// TIA Portal project "Divider LIE-09" (V14)

(* hardware
DEVICE "S7-1200 station"  S7-1200 Station
   slot 0: "Rack_0"  Rack  V1.0
   slot 1: "CLP_Divider"  CPU 1214C DC/DC/DC  6ES7 214-1AG40-0XB0  V4.1
   slot 2: "Analog_Output"  6ES7 232-4HD32-0XB0  V2.0
DEVICE "IHM_Divider"  KTP600 Basic mono PN
   slot 0: "HMI"  HMI  6AV6 647-0AB11-3AX0  12.0.0.0
   slot 1: "HMI_RT_2"  KTP600 Basic mono PN  6AV6 647-0AB11-3AX0  12.0.0.0
   slot 5: "IHM_Divider.IE_CP_1"  PROFINET Interface
      slot 1: "PROFINET Interface_1"  PROFINET Interface
         slot 1: "Port_1"  Port
*)

// ===== PLC "CLP_Divider"  CPU 1214C DC/DC/DC =====

VAR_GLOBAL   // PLC tag table "General"
   "Aux_Byte_0" AT %MB10 : Byte;
   "Aux_Byte_1" AT %MB11 : Byte;
   "Aux_Int" AT %MW10 : Int;
   "Aux_Real" AT %MD12 : Real;
   "Status Byte" AT %QB50 : Byte;   // Palavra de status enviada para a SteelBelt
END_VAR

VAR_GLOBAL   // PLC tag table "Digital Output"
   "DO - Ligar Inv 01" AT %Q0.0 : Bool;
   "DO - Ligar Inv 02" AT %Q0.1 : Bool;
   "DO - Reset Inv 01" AT %Q0.2 : Bool;
   "DO - Reset Inv 02" AT %Q0.3 : Bool;
   "DO - Ligar Inv Divider" AT %Q0.4 : Bool;
   "DO - Reserva 02" AT %Q0.5 : Bool;
   "DO - Reserva 03" AT %Q0.6 : Bool;
END_VAR

VAR_GLOBAL   // PLC tag table "Analog Input"
   "Divider Dancer Sensor" AT %IW100 : Int;
   "Potentiometer Jog" AT %IW102 : Int;
END_VAR

VAR_GLOBAL   // PLC tag table "System and Clock Memory"
   "Clock_0.5Hz" AT %M8191.7 : Bool;
   "Clock_0.625Hz" AT %M8191.6 : Bool;
   "Clock_1Hz" AT %M8191.5 : Bool;
   "Clock_1.25Hz" AT %M8191.4 : Bool;
   "Clock_2Hz" AT %M8191.3 : Bool;
   "Clock_2.5Hz" AT %M8191.2 : Bool;
   "Clock_5Hz" AT %M8191.1 : Bool;
   "Clock_10Hz" AT %M8191.0 : Bool;
   "Clock_Byte" AT %MB8191 : Byte;
   "AlwaysFALSE" AT %M8190.3 : Bool;
   "AlwaysTRUE" AT %M8190.2 : Bool;
   "DiagStatusUpdate" AT %M8190.1 : Bool;
   "FirstScan" AT %M8190.0 : Bool;
   "System_Byte" AT %MB8190 : Byte;
END_VAR

VAR_GLOBAL   // PLC tag table "Analog Output"
   "AO - Velocidade Inv 01" AT %QW100 : Int;
   "AO - Velocidade Inv 02" AT %QW102 : Int;
   "AO - Velocidade Divider" AT %QW106 : Int;
END_VAR

VAR_GLOBAL   // PLC tag table "Digital Input"
   "DI - Man/Auto" AT %I0.0 : Bool;
   "DI - Ligar Inv 01 Manual" AT %I0.1 : Bool;
   "DI - Ligar Inv 02 Manual" AT %I0.2 : Bool;
   "DI - Emergencia" AT %I0.3 : Bool;
   "DI - Liga\Desliga" AT %I0.4 : Bool;
   "DI - Falha Inversor 01" AT %I0.5 : Bool;
   "DI - Falha Inversor 02" AT %I0.6 : Bool;
   "DI - Botão JOG" AT %I0.7 : Bool;
   "DI - Reserva 02" AT %I1.0 : Bool;
   "DI - Reserva 03" AT %I1.1 : Bool;
END_VAR

VAR_GLOBAL   // PLC tag table "Fielbus"
   "Status Veloc. SteelBelt" AT %ID50 : Real;   // Valor recebido por rede da SteelBelt
   "Status Byte SteelBelt" AT %IB54 : Byte;   // Palavra de status recebida da SteelBelt
END_VAR

// folder: DB's

DATA_BLOCK "Status"   // DB1
{ S7_Optimized_Access := 'FALSE' }
VERSION : 0.1
   VAR
      "Velocidade SteelBelt" : Real;
      SteelBelt : Struct
         Parado : Bool;
         "Em operação" : Bool;
         "Emergência Ativa" : Bool;
         Falha : Bool;
         Manual : Bool;
         Automatico : Bool;
         "Spare 01" : Bool;
         Heartbeat : Bool;
      END_STRUCT;
      Divider : Struct
         Parado : Bool;
         "Em operação" : Bool;
         "Emergência Ativa" : Bool;
         "Falha Inv 01" : Bool;
         "Falha Inv 02" : Bool;
         Manual : Bool;
         Automatico : Bool;
         Heartbeat : Bool;
      END_STRUCT;
      "Fator %" : Real;
   END_VAR
BEGIN
END_DATA_BLOCK

DATA_BLOCK "DB_Controle"   // DB2
{ S7_Optimized_Access := 'TRUE' }
VERSION : 0.1
   VAR
      "Condições Auto" : Bool := FALSE;
      "Condições Manual" : Bool := FALSE;
      "Perda Comunicação" : Bool := TRUE;
      "Timer" : Array[1..10] of IEC_TIMER;
      "Reset Falha" : Bool := FALSE;
   END_VAR
BEGIN
   "Timer"[1].ST := T#0MS;
   "Timer"[1].PT := T#0MS;
   "Timer"[1].ET := T#0MS;
   "Timer"[1].RU := FALSE;
   "Timer"[1].IN := FALSE;
   "Timer"[1].Q := FALSE;
   "Timer"[2].ST := T#13D_17H_25M_16S_353MS;
   "Timer"[2].PT := T#500MS;
   "Timer"[2].ET := T#71MS;
   "Timer"[2].RU := TRUE;
   "Timer"[2].IN := TRUE;
   "Timer"[2].Q := FALSE;
   "Timer"[3].ST := T#13D_17H_25M_15S_851MS;
   "Timer"[3].PT := T#500MS;
   "Timer"[3].ET := T#0MS;
   "Timer"[3].RU := FALSE;
   "Timer"[3].IN := FALSE;
   "Timer"[3].Q := FALSE;
   "Timer"[4].ST := T#0MS;
   "Timer"[4].PT := T#0MS;
   "Timer"[4].ET := T#0MS;
   "Timer"[4].RU := FALSE;
   "Timer"[4].IN := FALSE;
   "Timer"[4].Q := FALSE;
   "Timer"[5].ST := T#2D_16H_45M_439MS;
   "Timer"[5].PT := T#2S;
   "Timer"[5].ET := T#2S;
   "Timer"[5].RU := FALSE;
   "Timer"[5].IN := TRUE;
   "Timer"[5].Q := TRUE;
   "Timer"[6].ST := T#0MS;
   "Timer"[6].PT := T#0MS;
   "Timer"[6].ET := T#0MS;
   "Timer"[6].RU := FALSE;
   "Timer"[6].IN := FALSE;
   "Timer"[6].Q := FALSE;
   "Timer"[7].ST := T#0MS;
   "Timer"[7].PT := T#0MS;
   "Timer"[7].ET := T#0MS;
   "Timer"[7].RU := FALSE;
   "Timer"[7].IN := FALSE;
   "Timer"[7].Q := FALSE;
   "Timer"[8].ST := T#0MS;
   "Timer"[8].PT := T#0MS;
   "Timer"[8].ET := T#0MS;
   "Timer"[8].RU := FALSE;
   "Timer"[8].IN := FALSE;
   "Timer"[8].Q := FALSE;
   "Timer"[9].ST := T#0MS;
   "Timer"[9].PT := T#0MS;
   "Timer"[9].ET := T#0MS;
   "Timer"[9].RU := FALSE;
   "Timer"[9].IN := FALSE;
   "Timer"[9].Q := FALSE;
   "Timer"[10].ST := T#0MS;
   "Timer"[10].PT := T#0MS;
   "Timer"[10].ET := T#0MS;
   "Timer"[10].RU := FALSE;
   "Timer"[10].IN := FALSE;
   "Timer"[10].Q := FALSE;
END_DATA_BLOCK

DATA_BLOCK "Divider Speed VFD"   // DB3
{ S7_Optimized_Access := 'TRUE' }
AUTHOR : Fernando
VERSION : 0.1
// stored: InstanceOfName Divider Speed
"Divider Speed"
BEGIN
END_DATA_BLOCK

DATA_BLOCK "DB_T_COMM"   // DB4
{ S7_Optimized_Access := 'TRUE' }
AUTHOR : Siemens
VERSION : 0.1
// stored: InstanceOfName T_COMM
"T_COMM"
BEGIN
END_DATA_BLOCK

DATA_BLOCK "DB_DATA"   // DB5
{ S7_Optimized_Access := 'TRUE' }
VERSION : 0.1
   VAR
      UserDataSend : Array[0..99] of Byte;   // User Data to send
      UserDataRec : Array[0..99] of Byte;   // User Data received
   END_VAR
   VAR RETAIN
      ServerIP : IP_V4;   // Server IP Address
      CommPort : UInt := 2849;
   END_VAR
BEGIN
   ServerIP.ADDR[1] := 192;
   ServerIP.ADDR[2] := 168;
   ServerIP.ADDR[3] := 1;
   ServerIP.ADDR[4] := 100;
END_DATA_BLOCK

DATA_BLOCK "Esteira 01"   // DB6
{ S7_Optimized_Access := 'TRUE' }
AUTHOR : Fernando
VERSION : 0.1
// stored: InstanceOfName Conveyor VFD
"Conveyor VFD"
BEGIN
END_DATA_BLOCK

DATA_BLOCK "Esteira 02"   // DB7
{ S7_Optimized_Access := 'TRUE' }
AUTHOR : Fernando
VERSION : 0.1
// stored: InstanceOfName Conveyor VFD
"Conveyor VFD"
BEGIN
END_DATA_BLOCK

DATA_BLOCK "Date Time"   // DB8
{ S7_Optimized_Access := 'TRUE' }
AUTHOR : Fernando
VERSION : 0.1
// stored: InstanceOfName Date and Time
"Date and Time"
BEGIN
END_DATA_BLOCK

DATA_BLOCK "HMI Area Pointer"   // DB100
TITLE = HMI AREA POINTER
{ S7_Optimized_Access := 'TRUE' }
AUTHOR : Fernando
VERSION : 0.1
   VAR
      Coordination : Word;
      DateTime : DTL;
      JobMailbox : Array[0..3] of Word;
      DataRecord : Array[0..4] of Word;
      ProjectID : Word;
      ScreenNumber : Array[0..4] of Word;
      DateTimePLC : Struct
         DateTime : DTL;
         Reserve_01 : Word;
         Reserve_02 : Word;
      END_STRUCT;
   END_VAR
BEGIN
END_DATA_BLOCK

// folder: (top level)

FUNCTION_BLOCK "T_COMM"   // FB1, SCL
TITLE = TCP communication function block
{ S7_Optimized_Access := 'TRUE' }
AUTHOR : Siemens
VERSION : 0.1
// Send and receive data over a TCP connection. Configurable as client or server and for sending and/or receiving data.
   VAR_INPUT
      Enable : Bool;   // Enable communication
      ConnId : Conn_Ouc;   // Connection ID
      InterfaceId : Hw_Any := 64;   // Interface ID
      ServerIP : IP_V4;   // Server IP Address
      CommPort : UInt;   // Port to be used for communication
      IsServer : Bool;   // Act as Server
      IsClient : Bool;   // Act as Client
      DataLen : UInt;   // Bytes to send / receive
      RecData : Bool;   // Enable receiving data
      SendData : Bool;   // Enable sending data
      Continuous : Bool := true;   // Continuous sending and receiving data
      WritePausePre : Time := T#1000ms;   // Pause between sending data
   END_VAR
   VAR_OUTPUT
      ConDn : Bool;   // Connected
      ConBusy : Bool;   // Waiting for connection
      Err : Bool;   // Collective error signal
   END_VAR
   VAR_IN_OUT
      DataSend : Array[0..99] of Byte;   // Byte array with user data to send
      DataRec : Array[0..99] of Byte;   // Byte array with user data received
   END_VAR
   VAR
      TCon : TCON;   // Establish communication connection
      TConParam : TCON_IP_v4;   // Connection parameters to establish communication connection
      TSend : TSEND;   // Send data via communication connection
      TRcv : TRCV;   // Receive data via communication connection
      TDiscon : TDISCON;   // Terminate communication connection
      TSendDnTof : TOF_TIME;   // Off-Delay Timer send done
      TSendDelay : Bool;   // Delay after sending active
      LocalEnable : Bool;   // Enable logic FB internal
      Reset : Bool;   // Reset communication
      Error : Bool;   // Error present
      Connected : Bool;   // Connection made
      Send1Time : Bool;   // Send data only one time
      Rec1Time : Bool;   // Receive data only one time
      TSendDn : Bool;   // Sending done
      TRcvNdr : Bool;   // New data received
      SingleDataPulse : Bool;   // Send / Receive one time - positive edge signal
      SingleDataMem : Bool;   // Send / Receive one time - positive edge signal memory bit
      SingleData : Bool;   // Send / Receive one time (continuous inverted)
      StatusWords : Struct   // Status words of communication instructions
         ConStatus : Word;   // Error status word of TCon
         SendStatus : Word;   // Error status word of TSend
         RcvStatus : Word;   // Error status word of TRcv
         DisconStatus : Word;   // Error status word of TDiscon
      END_STRUCT;
   END_VAR
   VAR_TEMP
      EnSend : Bool;   // Enable TSend instruction
      EnRcv : Bool;   // Enable TRcv instruction
      TConBusy : Bool;   // TCon busy status
      TConDn : Bool;   // TCon done status
      TConError : Bool;   // TCon error status
      TConStat : Word;   // TCon status word
      TSendBusy : Bool;   // TSend busy status
      TSendError : Bool;   // TSend error status
      TSendStatus : Word;   // TSend status word
      TRcvBusy : Bool;   // TRcv busy status
      TRcvError : Bool;   // TRcv error status
      TRcvStatus : Word;   // TRcv status word
      TRcvRcvdLen : UDInt;   // TRcv data length received
      TDisconError : Bool;   // TDiscon error status
      TDisconStatus : Word;   // TDiscon status word
   END_VAR
BEGIN
   //*** Connect Configuration
   #TConParam.InterfaceId := #InterfaceId;
   #TConParam.ID := #ConnId;
   #TConParam.ConnectionType := 11; //11 = TCP/IP
   #TConParam.ActiveEstablished := (#IsClient AND NOT #IsServer); //FALSE = Server; TRUE = Client
   #TConParam.RemoteAddress := #ServerIP;
   #TConParam.LocalPort := #CommPort;
   #TConParam.RemotePort := #TConParam.LocalPort;
   //*** End of connection configuration











   //Set a signal that data should be send and receive only one time
   #SingleData := #Enable AND NOT #Continuous;
   #SingleDataPulse := #SingleData AND NOT #SingleDataMem;
   #SingleDataMem := #SingleData;

   //Signal that data should only received one time (TRUE = receiving pending; FALSE = data received)
   #Rec1Time := #Enable AND ((#RecData AND #SingleDataPulse) OR (#Rec1Time AND NOT #TRcvNdr));
   //Signal that data should only send one time (TRUE = sending pending; FALSE = data sent)
   #Send1Time := #Enable AND ((#SendData AND #SingleDataPulse) OR (#Send1Time AND NOT #TSendDn));

   //Enable logic with enable input if other checks are OK
   #LocalEnable := #Enable AND NOT #Error AND (#Continuous OR #Rec1Time OR #Send1Time);

   //Enable Signal switched off
   #Reset := NOT #LocalEnable;

   //Connect
   #TCon(REQ := #LocalEnable,
         DONE => #TConDn,
         STATUS => #TConStat,
         BUSY => #TConBusy,
         ERROR => #TConError,
         CONNECT := #TConParam,
         ID := #TConParam.ID);
   //Connection status
   #Connected := #TConDn OR (#Connected AND #LocalEnable);

   //Enable TSEND instruction
   #EnSend := #Connected AND #SendData AND (#Send1Time OR #Continuous) AND NOT #TSendDelay;
   //Send data
   #TSend(ID := #TCon.ID,
          LEN := #DataLen,
          DATA := #DataSend,
          REQ := #EnSend,
          ERROR => #TSendError,
          STATUS => #TSendStatus,
          DONE => #TSendDn,
          BUSY => #TSendBusy);

   //Delay between sending data
   #TSendDnTof(IN := #TSendDn,
               PT := #WritePausePre,
               Q => #TSendDelay);

   //Enable TRCV instruction
   #EnRcv := #Connected AND #RecData AND (#Rec1Time OR #Continuous);
   //Receive data
   #TRcv(ID := #TCon.ID,
         LEN := #DataLen,
         DATA := #DataRec,
         ERROR => #TRcvError,
         EN_R := #EnRcv,
         STATUS => #TRcvStatus,
         NDR => #TRcvNdr,
         BUSY => #TRcvBusy,
         RCVD_LEN => #TRcvRcvdLen);






   // //Disconnect
   #TDiscon(ID := #TCon.ID,
            ERROR => #TDisconError,
            STATUS => #TDisconStatus,
            REQ := #Reset);

   //Fault signal - collect all fault from all T_ instructions
   #Error := (#TConError OR #TSendError OR #TRcvError OR #TDisconError) OR (#Error AND #Enable);

   //In case of error, store the status word
   IF #TConError THEN
       #StatusWords.ConStatus := #TConStat;
   END_IF;
   //In case of error, store the status word
   IF #TSendError THEN
       #StatusWords.SendStatus := #TSendStatus;
   END_IF;
   //In case of error, store the status word
   IF #TRcvError THEN
       #StatusWords.RcvStatus := #TRcvStatus;
   END_IF;
   //In case of error, store the status word
   IF #TDisconError THEN
       #StatusWords.DisconStatus := #TDisconStatus;
   END_IF;

   //Status Outputs
   #ConDn := #Connected;
   #Err := #Error;
   #ConBusy := #TConBusy;
END_FUNCTION_BLOCK

FUNCTION_BLOCK "Divider Speed"   // FB2, LAD
{ S7_Optimized_Access := 'TRUE' }
AUTHOR : Fernando
VERSION : 0.1
   VAR_OUTPUT
      "VFD Run" : Bool;
   END_VAR
   VAR
      "Divider Dancer" : "Input Analog";
      KEY_MARK : Bool;
   END_VAR
   VAR RETAIN
      "Check-mark" : Real;
   END_VAR
   VAR
      "Potentiometer Percent" : Real;
      "Divider Speed Boost" : Real;
      "Calculated Divider Speed Reference" : Real;
      "Divider Speed" : Real;
      "Run Auto" : Bool;
      "Run Manual" : Bool;
      Prototipar : Bool;
      Prototipagem : Bool;
      "Check-Mark_IHM" : Real;
      Temporizador : Array[0..10] of IEC_TIMER;
      tempo : Array[0..10] of Time;
   END_VAR
   VAR_TEMP
      Subtract : Real;
      Scale : Struct
         Potentiometer : Real;
         Divider : Real;
      END_STRUCT;
   END_VAR
   VAR CONSTANT
      "Divider Speed Factor Mutiplier" : Real := 0.12;
      NumberScreen : Int := 3;   // Tela número 03
   END_VAR
   VAR_TEMP   // added for the SCL form of the ladder/FBD networks
      _w1 : Bool;
   END_VAR
BEGIN

REGION Network 1: Potenciômetro para ajuste de velocidade do JOG
   // * Valor mínimo da saída: 5.0%
   // * Valor máximo da saída: 15.0%
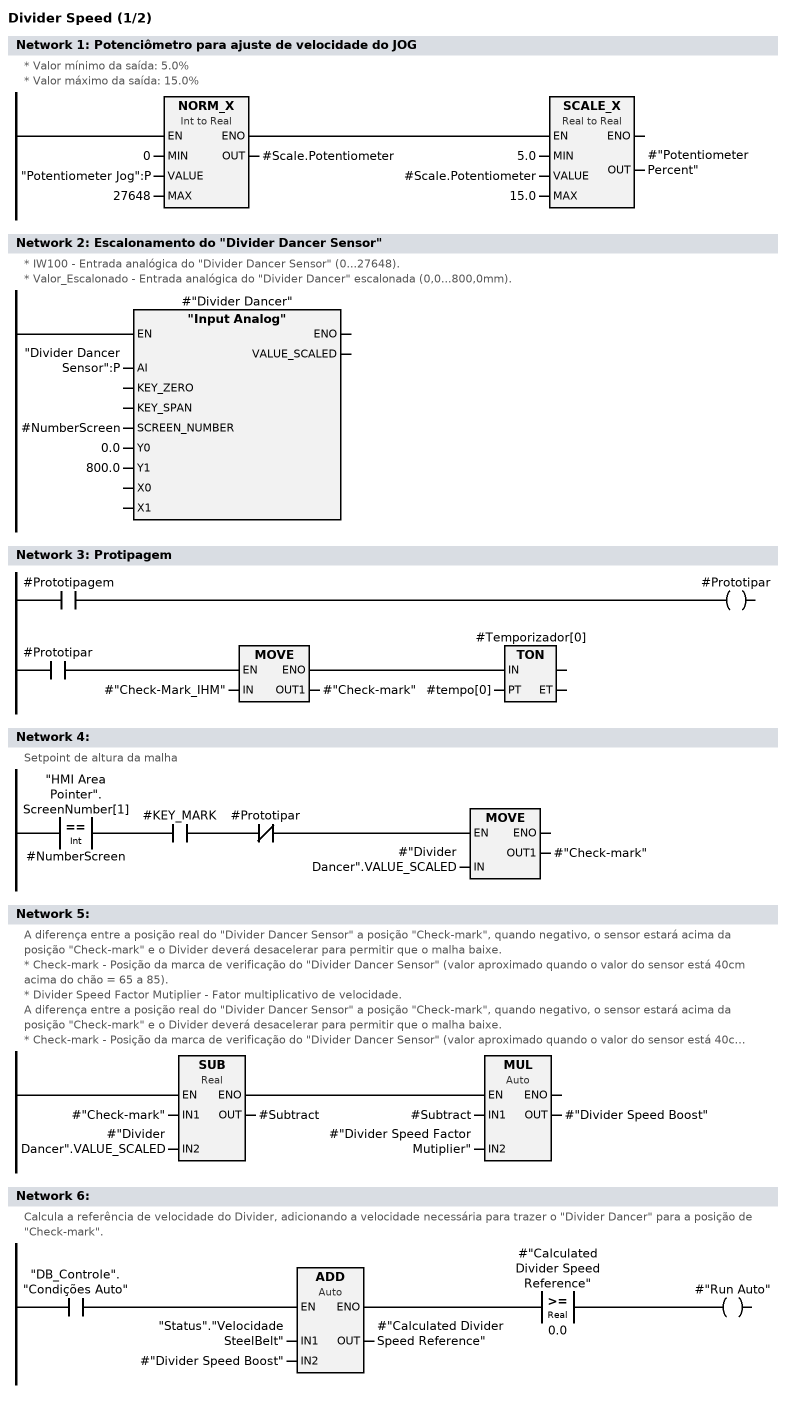
   RUNG wire#powerrail
      { S7_Templates := "[SrcType := Int, DestType := Real]" } Normalize(min := 0, value := "Potentiometer Jog":P, max := 27648, out => #Scale.Potentiometer)
      { S7_Templates := "[SrcType := Real, DestType := Real]" } Scale(min := 5.0, value := #Scale.Potentiometer, max := 15.0, out => #"Potentiometer Percent")
   END_RUNG
   // the same network as SCL:
   #Scale.Potentiometer := NORM_X(MIN := 0, VALUE := "Potentiometer Jog":P, MAX := 27648);
   #"Potentiometer Percent" := SCALE_X(MIN := 5.0, VALUE := #Scale.Potentiometer, MAX := 15.0);
END_REGION

REGION Network 2: Escalonamento do "Divider Dancer Sensor"
   // * IW100 - Entrada analógica do "Divider Dancer Sensor" (0...27648).
   // * Valor_Escalonado - Entrada analógica do "Divider Dancer" escalonada (0,0...800,0mm).
   RUNG wire#powerrail
      #"Divider Dancer"(AI := "Divider Dancer Sensor":P, KEY_ZERO :=, KEY_SPAN :=, SCREEN_NUMBER := #NumberScreen, Y0 := 0.0, Y1 := 800.0, X0 :=, X1 :=, VALUE_SCALED =>)
   END_RUNG
   // the same network as SCL:
   #"Divider Dancer"(AI := "Divider Dancer Sensor":P, SCREEN_NUMBER := #NumberScreen, Y0 := 0.0, Y1 := 800.0);   // "Input Analog"
END_REGION

REGION Network 3: Protipagem
   #Prototipar := #Prototipagem;
   IF #Prototipar THEN #"Check-mark" := #"Check-Mark_IHM"; END_IF;
   #Temporizador[0].TON(IN := #Prototipar, PT := #tempo[0]);
END_REGION

REGION Network 4
   // Setpoint de altura da malha
   RUNG wire#powerrail
      { S7_Templates := "SrcType := Int" } EQ_Contact(in1 := "HMI Area Pointer".ScreenNumber[1], in2 := #NumberScreen)
      Contact( #KEY_MARK )
      I_Contact( #Prototipar )
      Move(in := #"Divider Dancer".VALUE_SCALED, out1 => #"Check-mark")
   END_RUNG
   // the same network as SCL:
   IF ("HMI Area Pointer".ScreenNumber[1] = #NumberScreen) AND #KEY_MARK AND NOT #Prototipar THEN
       #"Check-mark" := #"Divider Dancer".VALUE_SCALED;
   END_IF;
END_REGION

REGION Network 5
   // A diferença entre a posição real do "Divider Dancer Sensor" a posição "Check-mark", quando negativo, o sensor estará acima da posição "Check-mark" e o Divider deverá desacelerar para permitir que o malha baixe.
   // 
   // * Check-mark - Posição da marca de verificação do "Divider Dancer Sensor" (valor aproximado quando o valor do sensor está 40cm acima do chão = 65 a 85).
   // * Divider Speed Factor Mutiplier - Fator multiplicativo de velocidade.
   // A diferença entre a posição real do "Divider Dancer Sensor" a posição "Check-mark", quando negativo, o sensor estará acima da posição "Check-mark" e o Divider deverá desacelerar para permitir que o malha baixe.
   // 
   // * Check-mark - Posição da marca de verificação do "Divider Dancer Sensor" (valor aproximado quando o valor do sensor está 40cm acima do chão).
   // * Divider Speed Factor Mutiplier - Fator multiplicativo de velocidade.
   RUNG wire#powerrail
      { S7_Templates := "SrcType := Real" } Sub(in1 := #"Check-mark", in2 := #"Divider Dancer".VALUE_SCALED, out => #Subtract)
      Mul(in1 := #Subtract, in2 := #"Divider Speed Factor Mutiplier", out => #"Divider Speed Boost")
   END_RUNG
   // the same network as SCL:
   #Subtract := #"Check-mark" - #"Divider Dancer".VALUE_SCALED;
   #"Divider Speed Boost" := #Subtract * #"Divider Speed Factor Mutiplier";
END_REGION

REGION Network 6
   // Calcula a referência de velocidade do Divider, adicionando a velocidade necessária para trazer o "Divider Dancer" para a posição de "Check-mark".
   RUNG wire#powerrail
      Contact( "DB_Controle"."Condições Auto" )
      Add(in1 := "Status"."Velocidade SteelBelt", in2 := #"Divider Speed Boost", out => #"Calculated Divider Speed Reference")
      { S7_Templates := "SrcType := Real" } GE_Contact(in1 := #"Calculated Divider Speed Reference", in2 := 0.0)
      Coil( #"Run Auto" )
   END_RUNG
   // the same network as SCL:
   IF "DB_Controle"."Condições Auto" THEN
       #"Calculated Divider Speed Reference" := "Status"."Velocidade SteelBelt" + #"Divider Speed Boost";
   END_IF;
   #"Run Auto" := "DB_Controle"."Condições Auto" AND (#"Calculated Divider Speed Reference" >= 0.0);
END_REGION

REGION Network 7
   // Em modo manual, a velocidade do Divider é definada pelo potenciômetro (JOG).
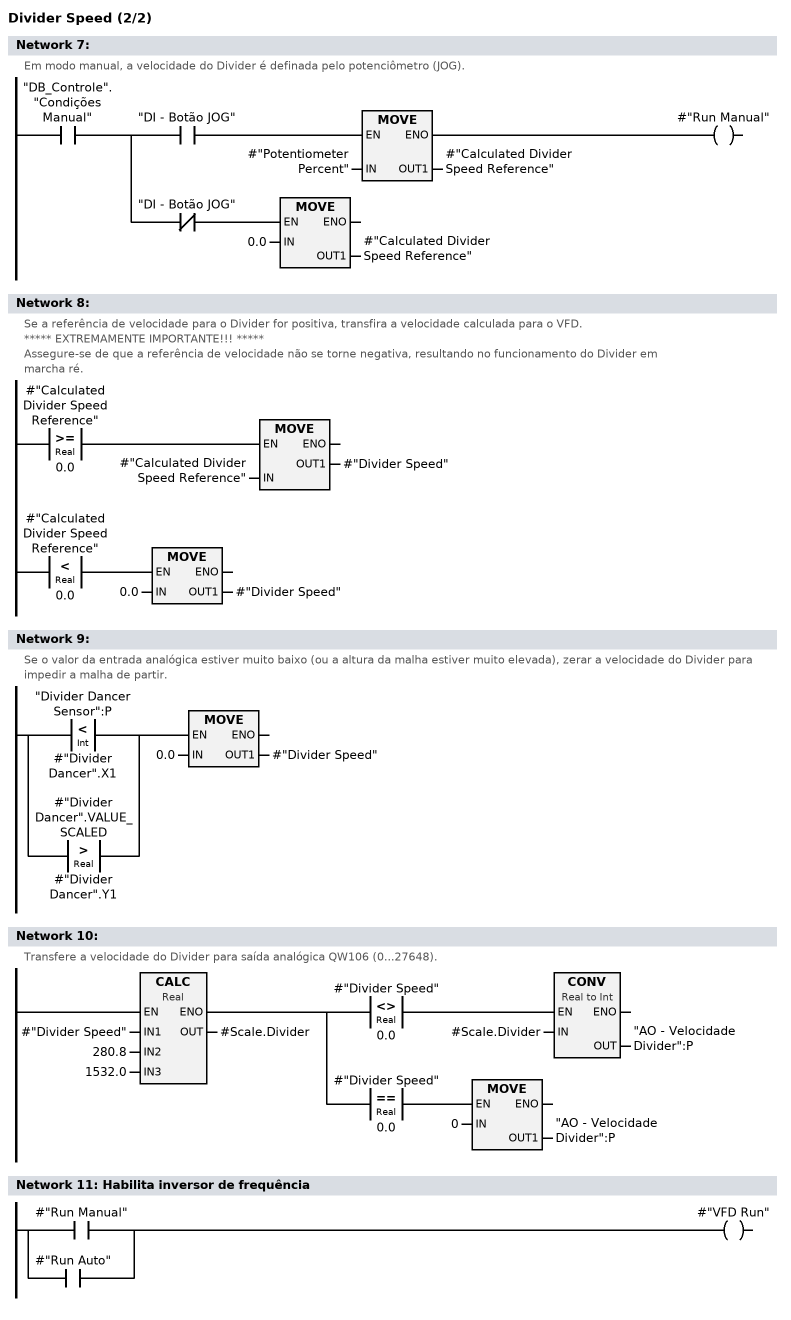
   RUNG wire#powerrail
      Contact( "DB_Controle"."Condições Manual" )
      wire#w1
      Contact( "DI - Botão JOG" )
      Move(in := #"Potentiometer Percent", out1 => #"Calculated Divider Speed Reference")
      Coil( #"Run Manual" )
   END_RUNG
   RUNG wire#w1
      I_Contact( "DI - Botão JOG" )
      Move(in := 0.0, out1 => #"Calculated Divider Speed Reference")
   END_RUNG
   // the same network as SCL:
   #_w1 := "DB_Controle"."Condições Manual" AND "DI - Botão JOG";
   IF #_w1 THEN #"Calculated Divider Speed Reference" := #"Potentiometer Percent"; END_IF;
   #"Run Manual" := #_w1;
   IF "DB_Controle"."Condições Manual" AND NOT "DI - Botão JOG" THEN
       #"Calculated Divider Speed Reference" := 0.0;
   END_IF;
END_REGION

REGION Network 8
   // Se a referência de velocidade para o Divider for positiva, transfira a velocidade calculada para o VFD.
   // 
   // ***** EXTREMAMENTE IMPORTANTE!!! *****
   // Assegure-se de que a referência de velocidade não se torne negativa, resultando no funcionamento do Divider em 
   // marcha ré.
   RUNG wire#powerrail
      { S7_Templates := "SrcType := Real" } GE_Contact(in1 := #"Calculated Divider Speed Reference", in2 := 0.0)
      Move(in := #"Calculated Divider Speed Reference", out1 => #"Divider Speed")
   END_RUNG
   RUNG wire#powerrail
      { S7_Templates := "SrcType := Real" } LT_Contact(in1 := #"Calculated Divider Speed Reference", in2 := 0.0)
      Move(in := 0.0, out1 => #"Divider Speed")
   END_RUNG
   // the same network as SCL:
   IF #"Calculated Divider Speed Reference" >= 0.0 THEN
       #"Divider Speed" := #"Calculated Divider Speed Reference";
   END_IF;
   IF #"Calculated Divider Speed Reference" < 0.0 THEN #"Divider Speed" := 0.0; END_IF;
END_REGION

REGION Network 9
   // Se o valor da entrada analógica estiver muito baixo (ou a altura da malha estiver muito elevada), zerar a velocidade do Divider para impedir a malha de partir.
   RUNG wire#powerrail
      { S7_Templates := "SrcType := Int" } LT_Contact(in1 := "Divider Dancer Sensor":P, in2 := #"Divider Dancer".X1)
      wire#w1
      Move(in := 0.0, out1 => #"Divider Speed")
   END_RUNG
   RUNG wire#powerrail
      { S7_Templates := "SrcType := Real" } GT_Contact(in1 := #"Divider Dancer".VALUE_SCALED, in2 := #"Divider Dancer".Y1)
   END_RUNG wire#w1
   // the same network as SCL:
   IF ("Divider Dancer Sensor":P < #"Divider Dancer".X1) OR (#"Divider Dancer".VALUE_SCALED > #"Divider Dancer".Y1) THEN
       #"Divider Speed" := 0.0;
   END_IF;
END_REGION

REGION Network 10
   // Transfere a velocidade do Divider para saída analógica QW106 (0...27648).
   CALC(in1 := #"Divider Speed", in2 := 280.8, in3 := 1532.0, out => #Scale.Divider);
   IF #"Divider Speed" <> 0.0 THEN "AO - Velocidade Divider":P := REAL_TO_INT(#Scale.Divider); END_IF;
   IF #"Divider Speed" = 0.0 THEN "AO - Velocidade Divider":P := 0; END_IF;
END_REGION

REGION Network 11: Habilita inversor de frequência
   RUNG wire#powerrail
      Contact( #"Run Manual" )
      wire#w1
      Coil( #"VFD Run" )
   END_RUNG
   RUNG wire#powerrail
      Contact( #"Run Auto" )
   END_RUNG wire#w1
   // the same network as SCL:
   #"VFD Run" := #"Run Manual" OR #"Run Auto";
END_REGION
END_FUNCTION_BLOCK

FUNCTION_BLOCK "Conveyor VFD"   // FB3, LAD
{ S7_Optimized_Access := 'TRUE' }
AUTHOR : Fernando
VERSION : 0.1
   VAR_INPUT
      Manual : Bool;
      Fault : Bool;
      "Factor %" : Real := 1.0;
   END_VAR
   VAR_OUTPUT
      "VFD Reset" : Bool;
      "VFD Run" : Bool;
      "Setpoint Speed" : Word;
   END_VAR
   VAR
      Speed : Real;
      "Speed Reference" : Real;
      "Speed Scaled" : Real;
      "Run Auto" : Bool;
      "Run Manual" : Bool;
      Ramp_Down : TOF_TIME;
   END_VAR
   VAR_TEMP
      Scale : Real;
   END_VAR
BEGIN

REGION Network 1
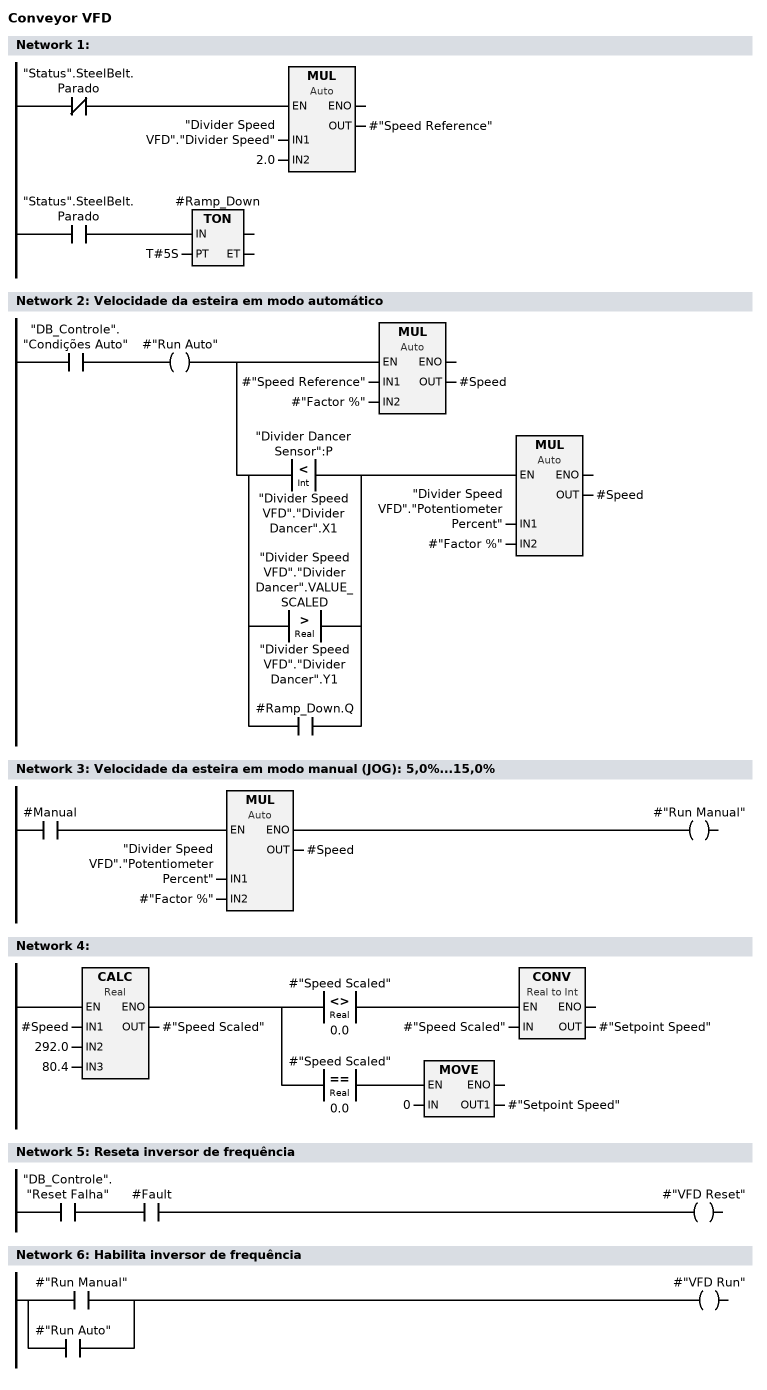
   IF NOT "Status".SteelBelt.Parado THEN
       #"Speed Reference" := "Divider Speed VFD"."Divider Speed" * 2.0;
   END_IF;
   #Ramp_Down(IN := "Status".SteelBelt.Parado, PT := T#5S);   // TON
END_REGION

REGION Network 2: Velocidade da esteira em modo automático
   RUNG wire#powerrail
      Contact( "DB_Controle"."Condições Auto" )
      Coil( #"Run Auto" )
      wire#w1
      Mul(in1 := #"Speed Reference", in2 := #"Factor %", out => #Speed)
   END_RUNG
   RUNG wire#w1
      { S7_Templates := "SrcType := Int" } LT_Contact(in1 := "Divider Dancer Sensor":P, in2 := "Divider Speed VFD"."Divider Dancer".X1)
      wire#w2
      Mul(in1 := "Divider Speed VFD"."Potentiometer Percent", in2 := #"Factor %", out => #Speed)
   END_RUNG
   RUNG wire#w1
      { S7_Templates := "SrcType := Real" } GT_Contact(in1 := "Divider Speed VFD"."Divider Dancer".VALUE_SCALED, in2 := "Divider Speed VFD"."Divider Dancer".Y1)
   END_RUNG wire#w2
   RUNG wire#w1
      Contact( #Ramp_Down.Q )
   END_RUNG wire#w2
   // the same network as SCL:
   #"Run Auto" := "DB_Controle"."Condições Auto";
   IF "DB_Controle"."Condições Auto" THEN #Speed := #"Speed Reference" * #"Factor %"; END_IF;
   IF "DB_Controle"."Condições Auto" AND (("Divider Dancer Sensor":P < "Divider Speed VFD"."Divider Dancer".X1) OR ("Divider Speed VFD"."Divider Dancer".VALUE_SCALED > "Divider Speed VFD"."Divider Dancer".Y1) OR #Ramp_Down.Q) THEN
       #Speed := "Divider Speed VFD"."Potentiometer Percent" * #"Factor %";
   END_IF;
END_REGION

REGION Network 3: Velocidade da esteira em modo manual (JOG): 5,0%...15,0%
   RUNG wire#powerrail
      Contact( #Manual )
      Mul(in1 := "Divider Speed VFD"."Potentiometer Percent", in2 := #"Factor %", out => #Speed)
      Coil( #"Run Manual" )
   END_RUNG
   // the same network as SCL:
   IF #Manual THEN #Speed := "Divider Speed VFD"."Potentiometer Percent" * #"Factor %"; END_IF;
   #"Run Manual" := #Manual;
END_REGION

REGION Network 4
   CALC(in1 := #Speed, in2 := 292.0, in3 := 80.4, out => #"Speed Scaled");
   IF #"Speed Scaled" <> 0.0 THEN #"Setpoint Speed" := REAL_TO_INT(#"Speed Scaled"); END_IF;
   IF #"Speed Scaled" = 0.0 THEN #"Setpoint Speed" := 0; END_IF;
END_REGION

REGION Network 5: Reseta inversor de frequência
   RUNG wire#powerrail
      Contact( "DB_Controle"."Reset Falha" )
      Contact( #Fault )
      Coil( #"VFD Reset" )
   END_RUNG
   // the same network as SCL:
   #"VFD Reset" := "DB_Controle"."Reset Falha" AND #Fault;
END_REGION

REGION Network 6: Habilita inversor de frequência
   RUNG wire#powerrail
      Contact( #"Run Manual" )
      wire#w1
      Coil( #"VFD Run" )
   END_RUNG
   RUNG wire#powerrail
      Contact( #"Run Auto" )
   END_RUNG wire#w1
   // the same network as SCL:
   #"VFD Run" := #"Run Manual" OR #"Run Auto";
END_REGION
END_FUNCTION_BLOCK

FUNCTION_BLOCK "Date and Time"   // FB4, SCL
{ S7_Optimized_Access := 'TRUE' }
AUTHOR : Fernando
VERSION : 0.1
   VAR_INPUT
      Screen : Int;
      ScreenNumber : Int;
   END_VAR
   VAR_IN_OUT
      DateTimeFromPLC : DTL;
   END_VAR
   VAR
      EditDateTime : Bool;
      ScreenEditHMI : Bool;
      DateTimeHMI : Struct
         YEAR : UInt;
         MONTH : USInt;
         DAY : USInt;
         HOUR : USInt;
         MINUTE : USInt;
         SECOND : USInt;
      END_STRUCT;
      R_TRIG : R_TRIG;
   END_VAR
   VAR_TEMP
      RetVal_RD : Int;
      RetVal_WR : Int;
   END_VAR
BEGIN
   //FERNANDO JÚNIOR
   //CRIADO: 24-06-2021

   REGION LEITURA DE DATA E HORA
       IF NOT #EditDateTime THEN
           #RetVal_RD := RD_SYS_T(#DateTimeFromPLC); //Lê a data e a hora do CLP.
       END_IF;
   END_REGION

   REGION TELA DE EDIÇÃO DE DATA E HORA
       IF (#Screen = #ScreenNumber) THEN //Tela de edição de data e hora da IHM.
           #ScreenEditHMI := TRUE;
       ELSE
           #ScreenEditHMI := FALSE;
       END_IF;

       #R_TRIG(CLK := #ScreenEditHMI); //Sinal da borda de subida.

       (*Ao acessar a tela de edição de data e hora da IHM,
       a data e hora atuais são transferidos para os campos de edição.*)
       IF #R_TRIG.Q THEN
           #DateTimeHMI.DAY := #DateTimeFromPLC.DAY;
           #DateTimeHMI.MONTH := #DateTimeFromPLC.MONTH;
           #DateTimeHMI.YEAR := #DateTimeFromPLC.YEAR;
           #DateTimeHMI.HOUR := #DateTimeFromPLC.HOUR;
           #DateTimeHMI.MINUTE := #DateTimeFromPLC.MINUTE;
           #DateTimeHMI.SECOND := #DateTimeFromPLC.SECOND;
       END_IF;
   END_REGION

   REGION EDIÇÃO DE DATA E HORA
       IF #EditDateTime THEN
           IF (#DateTimeHMI.DAY >= 1 & #DateTimeHMI.DAY <= 31) THEN //Valores entre 1 e 31 dias.
               #DateTimeFromPLC.DAY := #DateTimeHMI.DAY;
           END_IF;
           IF (#DateTimeHMI.MONTH >= 1 & #DateTimeHMI.MONTH <= 12) THEN //Valores entre 1 e 12 meses.
               #DateTimeFromPLC.MONTH := #DateTimeHMI.MONTH;
           END_IF;
           IF (#DateTimeHMI.YEAR >= 2020 & #DateTimeHMI.YEAR <= 3000) THEN //Valores a partir do ano 2020.
               #DateTimeFromPLC.YEAR := #DateTimeHMI.YEAR;
           END_IF;
           IF (#DateTimeHMI.HOUR >= 0 & #DateTimeHMI.HOUR <= 23) THEN //Valores entre 0 e 23 horas.
               #DateTimeFromPLC.HOUR := #DateTimeHMI.HOUR;
           END_IF;
           IF (#DateTimeHMI.MINUTE >= 0 & #DateTimeHMI.MINUTE <= 59) THEN //Valores entre 0 e 59 minutos.
               #DateTimeFromPLC.MINUTE := #DateTimeHMI.MINUTE;
           END_IF;
           IF (#DateTimeHMI.SECOND >= 0 & #DateTimeHMI.SECOND <= 59) THEN //Valores entre 0 e 59 segundos.
               #DateTimeFromPLC.SECOND := #DateTimeHMI.SECOND;
           END_IF;

           #DateTimeFromPLC.NANOSECOND := 0; //Ao editar o horário, será atribuido '0' aos nanosegundos. 

           #RetVal_WR := WR_SYS_T(#DateTimeFromPLC); //Escreve o horário no CLP.

       END_IF;
   END_REGION

   //FERNANDO JÚNIOR (fernando.junior@grupomoura.com)
   //24-06-2021
END_FUNCTION_BLOCK

FUNCTION_BLOCK "Input Analog"   // FB101, LAD
TITLE = INPUT ANALOG
{ S7_Optimized_Access := 'TRUE' }
AUTHOR : Fernando
VERSION : 0.1
// FERNANDO JÚNIOR (fernando.junior@grupomoura.com).
   VAR_INPUT
      AI : Word;   // Entrada Analógica
      KEY_ZERO : Bool;
      KEY_SPAN : Bool;
      SCREEN_NUMBER : Int;
      Y0 : Real := 0.0;
      Y1 : Real;
   END_VAR
   VAR_OUTPUT
      VALUE_SCALED : Real;
   END_VAR
   VAR_IN_OUT
      X0 : Int := 25550;
      X1 : Int := 910;
   END_VAR
   VAR
      Filtro : "Filter";
      Valor_Filtrado : Int;
      Calibrate : Struct   // Pulso para calibrar ZERO
         Zero : Bool;
         Span : Bool;
      END_STRUCT;
      Cal : Bool := FALSE;   // Pulso para executar calibração
      Escalonamento : "Scale";
      SignalEdge : Byte;
   END_VAR
   VAR_TEMP   // added for the SCL form of the ladder/FBD networks
      _w1 : Bool;
   END_VAR
BEGIN

REGION Network 1: FILTRO
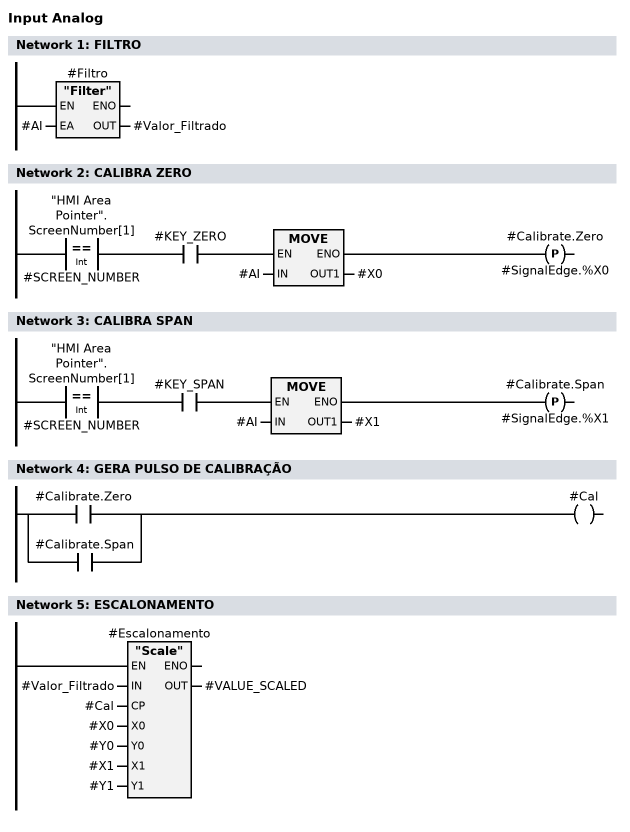
   RUNG wire#powerrail
      #Filtro(EA := #AI, OUT => #Valor_Filtrado)
   END_RUNG
   // the same network as SCL:
   #Filtro(EA := #AI, OUT => #Valor_Filtrado);   // "Filter"
END_REGION

REGION Network 2: CALIBRA ZERO
   #_w1 := ("HMI Area Pointer".ScreenNumber[1] = #SCREEN_NUMBER) AND #KEY_ZERO;
   IF #_w1 THEN #X0 := #AI; END_IF;
   #Calibrate.Zero := #_w1 AND NOT #SignalEdge.%X0;   // rising edge
   #SignalEdge.%X0 := #_w1;
END_REGION

REGION Network 3: CALIBRA SPAN
   #_w1 := ("HMI Area Pointer".ScreenNumber[1] = #SCREEN_NUMBER) AND #KEY_SPAN;
   IF #_w1 THEN #X1 := #AI; END_IF;
   #Calibrate.Span := #_w1 AND NOT #SignalEdge.%X1;   // rising edge
   #SignalEdge.%X1 := #_w1;
END_REGION

REGION Network 4: GERA PULSO DE CALIBRAÇÃO
   RUNG wire#powerrail
      Contact( #Calibrate.Zero )
      wire#w1
      Coil( #Cal )
   END_RUNG
   RUNG wire#powerrail
      Contact( #Calibrate.Span )
   END_RUNG wire#w1
   // the same network as SCL:
   #Cal := #Calibrate.Zero OR #Calibrate.Span;
END_REGION

REGION Network 5: ESCALONAMENTO
   RUNG wire#powerrail
      #Escalonamento(IN := #Valor_Filtrado, CP := #Cal, X0 := #X0, Y0 := #Y0, X1 := #X1, Y1 := #Y1, OUT => #VALUE_SCALED)
   END_RUNG
   // the same network as SCL:
   #Escalonamento(IN := #Valor_Filtrado,   // "Scale"
                  CP := #Cal,
                  X0 := #X0,
                  Y0 := #Y0,
                  X1 := #X1,
                  Y1 := #Y1,
                  OUT => #VALUE_SCALED);
END_REGION
END_FUNCTION_BLOCK

FUNCTION_BLOCK "Scale"   // FB102, SCL
TITLE = SCALE
{ S7_Optimized_Access := 'TRUE' }
AUTHOR : Fernando
VERSION : 0.1
   VAR_INPUT
      IN : Int;   // Valor efetivo da entrada
      CP : Bool := TRUE;   // Habilita cálculo dos fatores "M" e "B"
      X0 : Int;   // Valor inicial da abscissa X
      Y0 : Real;   // Valor inicial da ordenada Y
      X1 : Int;   // Valor final da abscissa X
      Y1 : Real;   // Valor final da ordenada Y
   END_VAR
   VAR_OUTPUT
      OUT : Real;   // Valor da saída calculada
   END_VAR
   VAR RETAIN
      "M" : Real := -0.03246753;   // Fator de escalonamento
   END_VAR
   VAR
      "B" : Real;   // Fator de offset
   END_VAR
BEGIN
   (*
   Gera uma saída linear em relação à entrada. Os parâmetros de entrada são:

   X0 = valor inicial do ponto X
   Y0 = valor inicial do ponto Y
   X1 = valor final do ponto X
   Y1 = valor final do ponto Y

   A fórmula para conversão da entrada é:

   OUT = (M * IN) + B

   Onde:

   OUT = saída
   M = fator de escalonamento = (Y1 - Y0) / (X1 - X0)
   IN = entrada
   B = offset = Y1 - (M * X1)

   Se a entrada CP estiver ligada, será feito o cálculo do valor de M, antes de calcular OUT, caso
   a entrada CP esteja desligada então será feito o cálculo de OUT com o último valor de M calculado.

   FERNANDO JÚNIOR
   CRIADO: 11-01-2021
   MODIFICADO: 21-05-2021
   *)

   REGION FATOR DE ESCALONAMENTO
       IF #CP THEN
           #"M" := (#Y1 - #Y0) / (#X1 - #X0);
       END_IF;
   END_REGION

   REGION OFFSET
       #"B" := #Y1 - (#"M" * #X1);
   END_REGION

   REGION OUTPUT
       #OUT := (#"M" * #IN) + #"B";
   END_REGION

   //FERNANDO JÚNIOR (fernando.junior@grupomoura.com).
   //21-05-2021
END_FUNCTION_BLOCK

FUNCTION_BLOCK "Filter"   // FB103, SCL
TITLE = FILTER
{ S7_Optimized_Access := 'TRUE' }
AUTHOR : Fernando
VERSION : 0.1
   VAR_INPUT
      EA : Int;   // Entrada Analógica
   END_VAR
   VAR_OUTPUT
      OUT : Int;   // Sinal Filtrado
   END_VAR
   VAR RETAIN
      INDEX_A : Int := 0;
      INDEX_B : Int := 0;
      INDEX_C : Int := 0;
      INDEX_D : Int := 0;
      SWAP : Int := 0;
      BUFFER : Array[0..30] of Int;
      ORDER : Array[0..30] of Int;
   END_VAR
   // BUFFER[1] := 0;
   // BUFFER[2] := 0;
   // BUFFER[3] := 0;
   // BUFFER[4] := 0;
   // BUFFER[5] := 0;
   // BUFFER[6] := 0;
   // BUFFER[7] := 0;
   // BUFFER[8] := 0;
   // BUFFER[9] := 0;
   // BUFFER[10] := 0;
BEGIN
   (*
   Classifica 31 amostras de uma variável de entrada, obtendo como resultado o valor da amostra central.

   Quando o bloco é chamado, o valor contido na entrada IN, será capturado como nova amostra e substituirá
   a amostra mais antiga. Em seguida será executada a classificação das amostras (valores das amostras em
   ordem crescente) e o valor da amostra central, após a classificação, será colocado na saída OUT (variável
   de saída do filtro).

   A primeira execução do bloco (após inicialização do CLP) preenche a pilha de amostras (buffer) e o valor
   da variável de saída OUT com o primeiro valor lido da variável de entrada IN.

   O BUFFER de armazenamento das amostras contem 31 elementos na pilha, sempre descartando o valor mais antigo
   da pilha e colocando em ordem crescente os valores.

   ##################################################
   IN -> Variável de entrada do filtro.
   OUT -> Variável de saída do filtro. Valor da amostra central (mediana).
   ##################################################

   FERNANDO JÚNIOR
   CRIAÇÃO: 14-01-2021
   MODIFICAÇÃO: 21-05-2021
   *)

   REGION ENTRADA ANALÓGICA
       (*
       BUFFER = ARMAZENA OS VALORES LIDOS NA
       ENTRADA ANALÓGICA A CADA CICLO DE SCAN.
       *)
       IF "FirstScan" THEN
           (*
           NO PRIMEIRO CICLO DE SCAN, A PRIMEIRA LEITURA
           DA ENTRADA ANALÓGICA É ESCRITA EM TODAS AS
           POSIÇÕES DO 'BUFFER'.
           *)
           FOR #INDEX_A := 0 TO 30 DO
               #BUFFER[#INDEX_A] := #EA;
           END_FOR;
       ELSE
           #BUFFER[#INDEX_A] := #EA;
       END_IF;
   END_REGION

   REGION VARIÁVEL DE ORDENAMENTO
       FOR #INDEX_B := 0 TO 30 DO
           #ORDER[#INDEX_B] := #BUFFER[#INDEX_B];
       END_FOR;
   END_REGION

   REGION ORDENA VALORES
       FOR #INDEX_C := 0 TO 30 DO
           FOR #INDEX_D := (#INDEX_C + 1) TO 30 DO
               IF (#ORDER[#INDEX_C] > #ORDER[#INDEX_D]) THEN
               (*
               COLOCA OS VALORES EM ORDEM CRESCENTE, PARA
               PODER ENCONTRAR A MEDIANA (VALOR CENTRAL).
               *)
                   #SWAP := #ORDER[#INDEX_C];
                   #ORDER[#INDEX_C] := #ORDER[#INDEX_D];
                   #ORDER[#INDEX_D] := #SWAP;
               END_IF;
           END_FOR;
       END_FOR;
   END_REGION

   REGION MEDIANA
       #OUT := #ORDER[(31/2)]; //VALOR CENTRAL.
   END_REGION

   REGION ZERA INDEXS
       IF (#INDEX_A < 30) THEN
           //INCREMENTA O VALOR DE 'INDEX_A'.
           #INDEX_A := #INDEX_A + 1;
       ELSE
           //ZERA O VALOR DE 'INDEX_A'.
           #INDEX_A := 0;
       END_IF;

       IF (#INDEX_B >= 30) THEN
           //ZERA O VALOR DE 'INDEX_B'.
           #INDEX_B := 0;
       END_IF;

       IF (#INDEX_C >= 30) THEN
           //ZERA O VALOR DE 'INDEX_C'.
           #INDEX_C := 0;
       END_IF;

       IF (#INDEX_D >= 30) THEN
           //ZERA O VALOR DE 'INDEX_D'.
           #INDEX_D := 0;
       END_IF;
   END_REGION

   //FERNANDO JÚNIOR (fernando.junior@grupomoura.com).
   //21-05-2021.
END_FUNCTION_BLOCK

FUNCTION "Comm Divider-SteelBelt" : Void   // FC1, LAD
{ S7_Optimized_Access := 'TRUE' }
VERSION : 0.1
   VAR_TEMP   // added for the SCL form of the ladder/FBD networks
      _w1 : Bool;
   END_VAR
BEGIN

REGION Network 1: Converte a velocidade da SteelBelt
   // MW10 = MB10 AND MB11
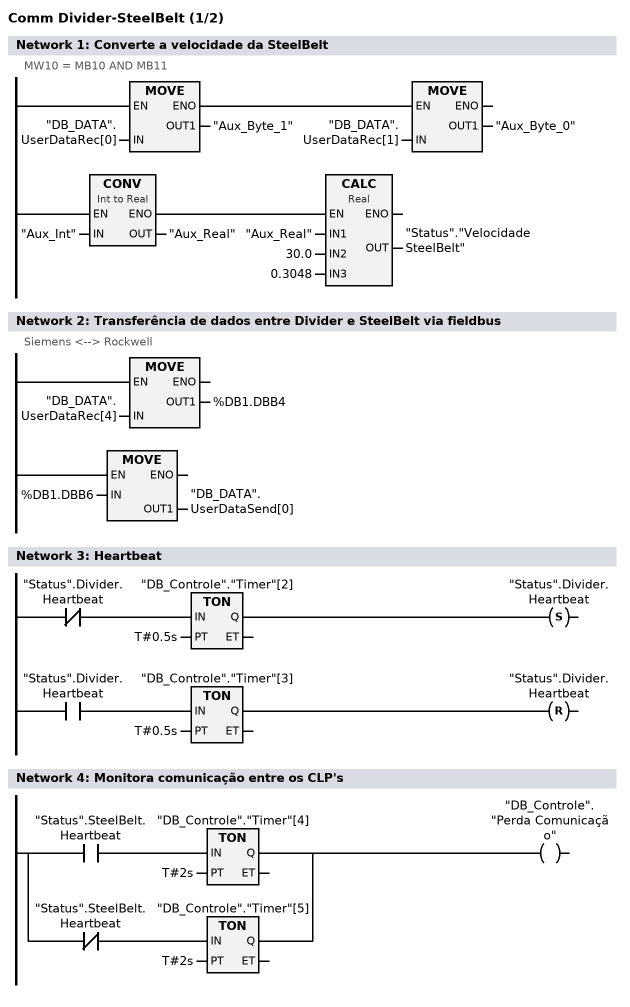
   "Aux_Byte_1" := "DB_DATA".UserDataRec[0];
   "Aux_Byte_0" := "DB_DATA".UserDataRec[1];
   "Aux_Real" := INT_TO_REAL("Aux_Int");
   CALC(in1 := "Aux_Real", in2 := 30.0, in3 := 0.3048, out => "Status"."Velocidade SteelBelt");
END_REGION

REGION Network 2: Transferência de dados entre Divider e SteelBelt via fieldbus
   // Siemens <--> Rockwell
   RUNG wire#powerrail
      Move(in := "DB_DATA".UserDataRec[4], out1 => %DB1.DBB4)
   END_RUNG
   RUNG wire#powerrail
      Move(in := %DB1.DBB6, out1 => "DB_DATA".UserDataSend[0])
   END_RUNG
   // the same network as SCL:
   %DB1.DBB4 := "DB_DATA".UserDataRec[4];
   "DB_DATA".UserDataSend[0] := %DB1.DBB6;
END_REGION

REGION Network 3: Heartbeat
   "DB_Controle"."Timer"[2].TON(IN := NOT "Status".Divider.Heartbeat, PT := T#0.5s);
   IF "DB_Controle"."Timer"[2].Q THEN "Status".Divider.Heartbeat := TRUE; END_IF;
   "DB_Controle"."Timer"[3].TON(IN := "Status".Divider.Heartbeat, PT := T#0.5s);
   IF "DB_Controle"."Timer"[3].Q THEN "Status".Divider.Heartbeat := FALSE; END_IF;
END_REGION

REGION Network 4: Monitora comunicação entre os CLP's
   "DB_Controle"."Timer"[4].TON(IN := "Status".SteelBelt.Heartbeat, PT := T#2s);
   #_w1 := "DB_Controle"."Timer"[4].Q;
   "DB_Controle"."Timer"[5].TON(IN := NOT "Status".SteelBelt.Heartbeat, PT := T#2s);
   "DB_Controle"."Perda Comunicação" := #_w1 OR "DB_Controle"."Timer"[5].Q;
END_REGION

REGION Network 5: Bloco de comunicação T_COMM
   // Siemens <--> Rockwell
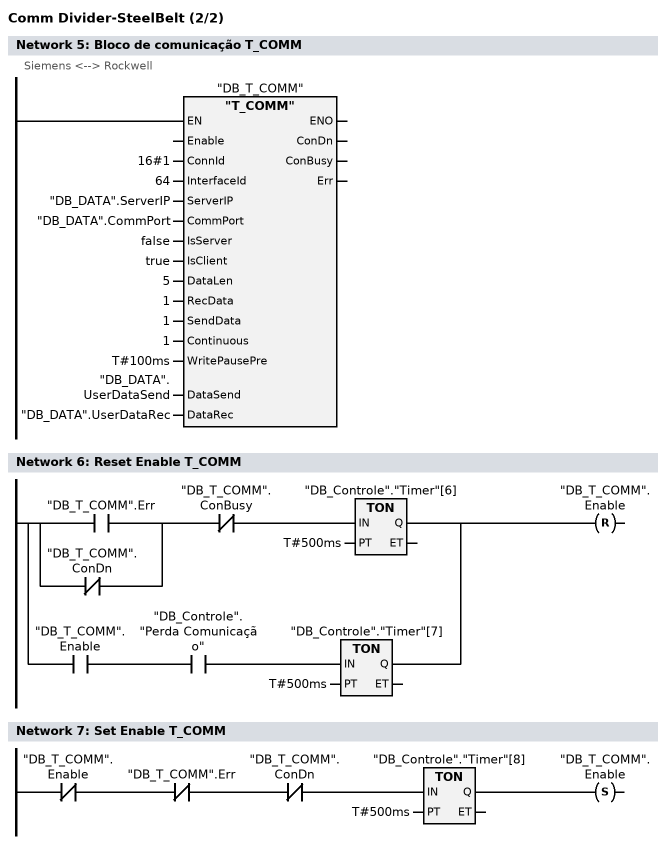
   RUNG wire#powerrail
      "DB_T_COMM"(Enable :=, ConnId := 16#1, InterfaceId := 64, ServerIP := "DB_DATA".ServerIP, CommPort := "DB_DATA".CommPort, IsServer := false, IsClient := true, DataLen := 5, RecData := 1, SendData := 1, Continuous := 1, WritePausePre := T#100ms, DataSend := "DB_DATA".UserDataSend, DataRec := "DB_DATA".UserDataRec, ConDn =>, ConBusy =>, Err =>)
   END_RUNG
   // the same network as SCL:
   "DB_T_COMM"(ConnId := 16#1,   // "T_COMM"
               InterfaceId := 64,
               ServerIP := "DB_DATA".ServerIP,
               CommPort := "DB_DATA".CommPort,
               IsServer := false,
               IsClient := true,
               DataLen := 5,
               RecData := 1,
               SendData := 1,
               Continuous := 1,
               WritePausePre := T#100ms,
               DataSend := "DB_DATA".UserDataSend,
               DataRec := "DB_DATA".UserDataRec);
END_REGION

REGION Network 6: Reset Enable T_COMM
   "DB_Controle"."Timer"[6].TON(IN := ("DB_T_COMM".Err OR NOT "DB_T_COMM".ConDn) AND NOT "DB_T_COMM".ConBusy,
                           PT := T#500ms);
   #_w1 := "DB_Controle"."Timer"[6].Q;
   "DB_Controle"."Timer"[7].TON(IN := "DB_T_COMM".Enable AND "DB_Controle"."Perda Comunicação", PT := T#500ms);
   IF #_w1 OR "DB_Controle"."Timer"[7].Q THEN "DB_T_COMM".Enable := FALSE; END_IF;
END_REGION

REGION Network 7: Set Enable T_COMM
   "DB_Controle"."Timer"[8].TON(IN := NOT "DB_T_COMM".Enable AND NOT "DB_T_COMM".Err AND NOT "DB_T_COMM".ConDn,
                           PT := T#500ms);
   IF "DB_Controle"."Timer"[8].Q THEN "DB_T_COMM".Enable := TRUE; END_IF;
END_REGION
END_FUNCTION

FUNCTION "Control" : Void   // FC2, LAD
{ S7_Optimized_Access := 'TRUE' }
VERSION : 0.1
   VAR_TEMP
      VFD : Struct   // Costantes da entrada analógica
         X0 : Word;
         X1 : Word;
      END_STRUCT;
      "Divider Speed Real" : Real;
      "Divider Speed Int" : Int;
   END_VAR
   VAR CONSTANT
      Fator : Real := 1.0;
   END_VAR
BEGIN

REGION Network 1: MANUAL / AUTOMÁTICO
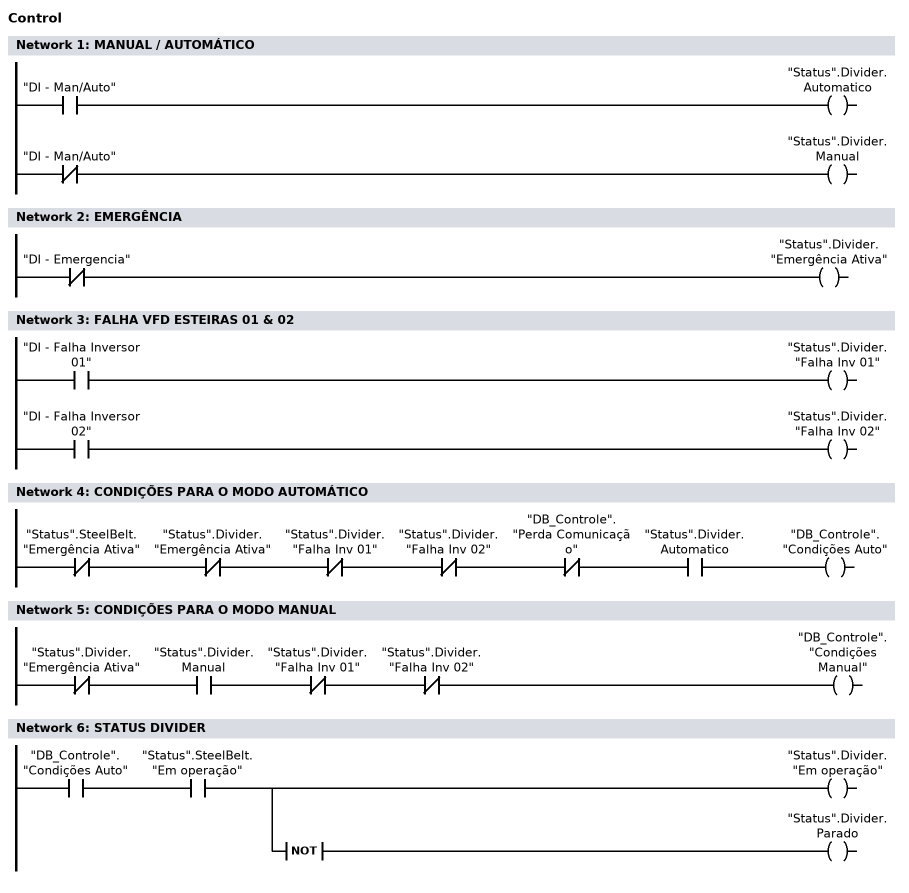
   RUNG wire#powerrail
      Contact( "DI - Man/Auto" )
      Coil( "Status".Divider.Automatico )
   END_RUNG
   RUNG wire#powerrail
      I_Contact( "DI - Man/Auto" )
      Coil( "Status".Divider.Manual )
   END_RUNG
   // the same network as SCL:
   "Status".Divider.Automatico := "DI - Man/Auto";
   "Status".Divider.Manual := NOT "DI - Man/Auto";
END_REGION

REGION Network 2: EMERGÊNCIA
   RUNG wire#powerrail
      I_Contact( "DI - Emergencia" )
      Coil( "Status".Divider."Emergência Ativa" )
   END_RUNG
   // the same network as SCL:
   "Status".Divider."Emergência Ativa" := NOT "DI - Emergencia";
END_REGION

REGION Network 3: FALHA VFD ESTEIRAS 01 & 02
   RUNG wire#powerrail
      Contact( "DI - Falha Inversor 01" )
      Coil( "Status".Divider."Falha Inv 01" )
   END_RUNG
   RUNG wire#powerrail
      Contact( "DI - Falha Inversor 02" )
      Coil( "Status".Divider."Falha Inv 02" )
   END_RUNG
   // the same network as SCL:
   "Status".Divider."Falha Inv 01" := "DI - Falha Inversor 01";
   "Status".Divider."Falha Inv 02" := "DI - Falha Inversor 02";
END_REGION

REGION Network 4: CONDIÇÕES PARA O MODO AUTOMÁTICO
   RUNG wire#powerrail
      I_Contact( "Status".SteelBelt."Emergência Ativa" )
      I_Contact( "Status".Divider."Emergência Ativa" )
      I_Contact( "Status".Divider."Falha Inv 01" )
      I_Contact( "Status".Divider."Falha Inv 02" )
      I_Contact( "DB_Controle"."Perda Comunicação" )
      Contact( "Status".Divider.Automatico )
      Coil( "DB_Controle"."Condições Auto" )
   END_RUNG
   // the same network as SCL:
   "DB_Controle"."Condições Auto" := NOT "Status".SteelBelt."Emergência Ativa" AND NOT "Status".Divider."Emergência Ativa" AND NOT "Status".Divider."Falha Inv 01" AND NOT "Status".Divider."Falha Inv 02" AND NOT "DB_Controle"."Perda Comunicação" AND "Status".Divider.Automatico;
END_REGION

REGION Network 5: CONDIÇÕES PARA O MODO MANUAL
   RUNG wire#powerrail
      I_Contact( "Status".Divider."Emergência Ativa" )
      Contact( "Status".Divider.Manual )
      I_Contact( "Status".Divider."Falha Inv 01" )
      I_Contact( "Status".Divider."Falha Inv 02" )
      Coil( "DB_Controle"."Condições Manual" )
   END_RUNG
   // the same network as SCL:
   "DB_Controle"."Condições Manual" := NOT "Status".Divider."Emergência Ativa" AND "Status".Divider.Manual AND NOT "Status".Divider."Falha Inv 01" AND NOT "Status".Divider."Falha Inv 02";
END_REGION

REGION Network 6: STATUS DIVIDER
   RUNG wire#powerrail
      Contact( "DB_Controle"."Condições Auto" )
      Contact( "Status".SteelBelt."Em operação" )
      wire#w1
      Coil( "Status".Divider."Em operação" )
   END_RUNG
   RUNG wire#w1
      Not()
      Coil( "Status".Divider.Parado )
   END_RUNG
   // the same network as SCL:
   "Status".Divider."Em operação" := "DB_Controle"."Condições Auto" AND "Status".SteelBelt."Em operação";
   "Status".Divider.Parado := NOT "Status".Divider."Em operação";
END_REGION
END_FUNCTION

ORGANIZATION_BLOCK "Main"   // OB1, LAD, ProgramCycle
TITLE = "Main Program Sweep (Cycle)"
{ S7_Optimized_Access := 'TRUE' }
VERSION : 0.1
   VAR_INPUT
      Initial_Call : Bool;   // Initial call of this OB
      Remanence : Bool;   // =True, if remanent data are available
   END_VAR
   VAR CONSTANT
      DateTimeScreen : Int := 6;   // Tela número 06
   END_VAR
BEGIN

REGION Network 1: Transferência de dados entre Divider e SteelBelt via fieldbus
   // Siemens <--> Rockwell.
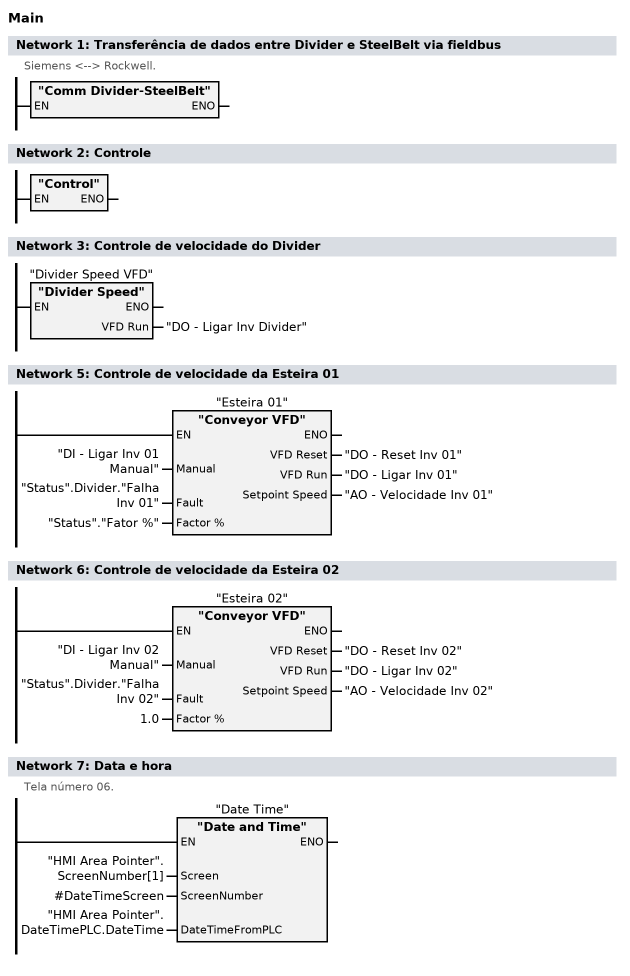
   RUNG wire#powerrail
      "Comm Divider-SteelBelt"()
   END_RUNG
   // the same network as SCL:
   "Comm Divider-SteelBelt"();
END_REGION

REGION Network 2: Controle
   RUNG wire#powerrail
      "Control"()
   END_RUNG
   // the same network as SCL:
   "Control"();
END_REGION

REGION Network 3: Controle de velocidade do Divider
   RUNG wire#powerrail
      "Divider Speed VFD"("VFD Run" => "DO - Ligar Inv Divider")
   END_RUNG
   // the same network as SCL:
   "Divider Speed VFD"("VFD Run" => "DO - Ligar Inv Divider");   // "Divider Speed"
END_REGION

REGION Network 4 (SCL): Limites do fator multiplicativo (1,0...2.0)
   IF "Status"."Fator %" < 1.0 THEN
       "Status"."Fator %" := 1.0;
   END_IF;
   IF "Status"."Fator %" > 2.0 THEN
       "Status"."Fator %" := 2.0;
   END_IF;
END_REGION

REGION Network 5: Controle de velocidade da Esteira 01
   RUNG wire#powerrail
      "Esteira 01"(Manual := "DI - Ligar Inv 01 Manual", Fault := "Status".Divider."Falha Inv 01", "Factor %" := "Status"."Fator %", "VFD Reset" => "DO - Reset Inv 01", "VFD Run" => "DO - Ligar Inv 01", "Setpoint Speed" => "AO - Velocidade Inv 01")
   END_RUNG
   // the same network as SCL:
   "Esteira 01"(Manual := "DI - Ligar Inv 01 Manual",   // "Conveyor VFD"
                Fault := "Status".Divider."Falha Inv 01",
                "Factor %" := "Status"."Fator %",
                "VFD Reset" => "DO - Reset Inv 01",
                "VFD Run" => "DO - Ligar Inv 01",
                "Setpoint Speed" => "AO - Velocidade Inv 01");
END_REGION

REGION Network 6: Controle de velocidade da Esteira 02
   RUNG wire#powerrail
      "Esteira 02"(Manual := "DI - Ligar Inv 02 Manual", Fault := "Status".Divider."Falha Inv 02", "Factor %" := 1.0, "VFD Reset" => "DO - Reset Inv 02", "VFD Run" => "DO - Ligar Inv 02", "Setpoint Speed" => "AO - Velocidade Inv 02")
   END_RUNG
   // the same network as SCL:
   "Esteira 02"(Manual := "DI - Ligar Inv 02 Manual",   // "Conveyor VFD"
                Fault := "Status".Divider."Falha Inv 02",
                "Factor %" := 1.0,
                "VFD Reset" => "DO - Reset Inv 02",
                "VFD Run" => "DO - Ligar Inv 02",
                "Setpoint Speed" => "AO - Velocidade Inv 02");
END_REGION

REGION Network 7: Data e hora
   // Tela número 06.
   RUNG wire#powerrail
      "Date Time"(Screen := "HMI Area Pointer".ScreenNumber[1], ScreenNumber := #DateTimeScreen, DateTimeFromPLC := "HMI Area Pointer".DateTimePLC.DateTime)
   END_RUNG
   // the same network as SCL:
   "Date Time"(Screen := "HMI Area Pointer".ScreenNumber[1],   // "Date and Time"
               ScreenNumber := #DateTimeScreen,
               DateTimeFromPLC := "HMI Area Pointer".DateTimePLC.DateTime);
END_REGION

REGION Network 8 (SCL): *** Info ***
   (*----------------------------------------
   Acumuladores Moura S.A. (Un. 01)
   Energia e Automação
   Fernando Júnior
   28-01-2023
   ----------------------------------------*)
END_REGION
END_ORGANIZATION_BLOCK

(* ===== HMI "HMI_RT_2" =====
system functions are stored by id; their names below are inferred from use
connection "HMI_DIVIDER": ETHERNET, SMART_S7_1200_OMS

HMI tags "Default tag table"
   "Status_Velocidade SteelBelt" : Real = PLC Status."Velocidade SteelBelt" AT %DB1.DBD0, 100 ms
   "Status_Diverger.Em operação" : Bool = PLC Status.Divider."Em operação" AT %DB1.DBX6.1, 1 s
   "Status_Diverger.Emergência Ativa" : Bool = PLC Status.Divider."Emergência Ativa" AT %DB1.DBX6.2, 1 s
   "Status_Diverger.Manual" : Bool = PLC Status.Divider.Manual AT %DB1.DBX6.5, 1 s
   "Status_Diverger.Falha Inv 01" : Bool = PLC Status.Divider."Falha Inv 01" AT %DB1.DBX6.3, 1 s
   "Status_Diverger.Falha Inv 02" : Bool = PLC Status.Divider."Falha Inv 02" AT %DB1.DBX6.4, 1 s
   "Status_Empastadeira.Em operação" : Bool = PLC Status.SteelBelt."Em operação" AT %DB1.DBX4.1, 1 s
   "Status_Empastadeira.Emergência Ativa" : Bool = PLC Status.SteelBelt."Emergência Ativa" AT %DB1.DBX4.2, 1 s
   "Status_Empastadeira.Manual" : Bool = PLC Status.SteelBelt.Manual AT %DB1.DBX4.4, 1 s
   "Status_Empastadeira.Automatico" : Bool = PLC Status.SteelBelt.Automatico AT %DB1.DBX4.5, 1 s
   "Status_Empastadeira.Heartbeat" : Bool = PLC Status.SteelBelt.Heartbeat AT %DB1.DBX4.7, 1 s
   "DB_Controle_Reset Falha" : Bool = PLC DB_Controle."Reset Falha", 1 s
   "DB_Controle_Perda Comunicação" : Bool = PLC DB_Controle."Perda Comunicação", 1 s
   "Status_Diverger.Automatico" : Bool = PLC Status.Divider.Automatico AT %DB1.DBX6.6, 1 s
   "Esteira 01_Speed" : Real = PLC "Esteira 01".Speed, 1 s
   "Esteira 02_Speed" : Real = PLC "Esteira 02".Speed, 1 s
   "Status_Fator %" : Real = PLC Status."Fator %" AT %DB1.DBD8, 1 s

HMI tags "Date and Time"
   "Ano" : UInt = PLC "Date Time".DateTimeHMI.YEAR, 1 s
   "Dia" : USInt = PLC "Date Time".DateTimeHMI.DAY, 1 s
   "Hora" : USInt = PLC "Date Time".DateTimeHMI.HOUR, 1 s
   "Mês" : USInt = PLC "Date Time".DateTimeHMI.MONTH, 1 s
   "Minuto" : USInt = PLC "Date Time".DateTimeHMI.MINUTE, 1 s
   "Segundo" : USInt = PLC "Date Time".DateTimeHMI.SECOND, 1 s
   "Editar_Data_Hora" : Bool = PLC "Date Time".EditDateTime, 1 s

HMI tags "Digital Input"
   "I0.0 - MAN / AUTO" : Bool = PLC "DI - Man/Auto" AT %I0.0, 1 s
   "I0.1 - VFD 01 MANUAL" : Bool = PLC "DI - Ligar Inv 01 Manual" AT %I0.1, 1 s
   "I0.2 - VFD 02 MANUAL" : Bool = PLC "DI - Ligar Inv 02 Manual" AT %I0.2, 1 s
   "I0.3 - EMERGÊNCIA" : Bool = PLC "DI - Emergencia" AT %I0.3, 1 s
   "I0.4 - LIGA / DESLIGA" : Bool = PLC "DI - Liga\Desliga" AT %I0.4, 1 s
   "I0.5 - FALHA VFD 01" : Bool = PLC "DI - Falha Inversor 01" AT %I0.5, 1 s
   "I0.6 - FALHA VFD 02" : Bool = PLC "DI - Falha Inversor 02" AT %I0.6, 1 s
   "I0.7 - BOTÃO JOG" : Bool = PLC "DI - Botão JOG" AT %I0.7, 1 s

HMI tags "Digital Output"
   "Q0.0 - LIGA VFD 01" : Bool = PLC "DO - Ligar Inv 01" AT %Q0.0, 1 s
   "Q0.1 - LIGA VFD 02" : Bool = PLC "DO - Ligar Inv 02" AT %Q0.1, 1 s
   "Q0.2 - RESET VFD 01" : Bool = PLC "DO - Reset Inv 01" AT %Q0.2, 1 s
   "Q0.3 - RESET VFD 02" : Bool = PLC "DO - Reset Inv 02" AT %Q0.3, 1 s
   "Q0.4 - LIGA VFD DIVIDER" : Bool = PLC "DO - Ligar Inv Divider" AT %Q0.4, 1 s

HMI tags "Internal Tags"
   "Número da Tela" : SInt, internal
   "Sempre_0" : SInt, internal
   "Pop-up SPAN" : Bool, internal
   "Pop-up ZERO" : Bool, internal

HMI tags "Divider"
   "Check_mark" : Real = PLC "Divider Speed VFD".Check-mark, 1 s
   "KEY_SPAN" : Bool = PLC "Divider Speed VFD"."Divider Dancer".KEY_SPAN, 1 s
   "KEY_ZERO" : Bool = PLC "Divider Speed VFD"."Divider Dancer".KEY_ZERO, 1 s
   "Sensor_Escalonado" : Real = PLC "Divider Speed VFD"."Divider Dancer".VALUE_SCALED, 1 s
   "Divider Dancer.X0" : Int = PLC "Divider Speed VFD"."Divider Dancer".X0, 1 s
   "Divider Dancer.X1" : Int = PLC "Divider Speed VFD"."Divider Dancer".X1, 1 s
   "KEY_MARK" : Bool = PLC "Divider Speed VFD".KEY_MARK, 1 s
   "Divider Speed" : Real = PLC "Divider Speed VFD"."Divider Speed", 1 s
   "Prototipagem" : Bool = PLC "Divider Speed VFD".Prototipagem AT %DB1.DBX0.0, 1 s
   "Check-mark_IHM" : Real = PLC "Divider Speed VFD".Check-Mark_IHM AT %DB1.DBD0, 1 s

text list "Mês": 1 'Janeiro'; 2 'Fevereiro'; 3 'Março'; 4 'Abril'; 5 'Maio'; 6 'Junho'; 7 'Julho'; 8 'Agosto'; 9 'Setembro'; 10 'Outubro'; 11 'Novembro'; 12 'Dezembro'; 0 'Mês'

text list "NomeTela": 1 'INÍCIO'; 2 'MENU'; 4 'ENTRADAS'; 5 'SAÍDAS'; 3 'VELOCIDADES'; 6 'DATA E HORA'; 7 'NomeTela'

Template "MOURA" 320x240
   GraphicView "Logo_Moura" at 2,3 size 76x24; Picture "Moura"
   Group "Gp_Títulos" at 85,5 size 150x20; TextList "NomeTela"
   Group "Data_Hora" at 240,0 size 76x30
   SymbolicIOField "Nome Tela" at 85,5 size 150x20; TextOn '1'; TextOff '0'; TextList "NomeTela"
      ProcessValue <- "Número da Tela"
   Group "Gp_BarraTítulos" at 0,0 size 320x30; Picture "Moura"; TextList "NomeTela"
   DateTimeField "Hora" at 240,12 size 76x18
   DateTimeField "Data" at 240,0 size 75x18
   Group "Data e Hora" at 240,0 size 76x30
   Button "Botão_DataHora" at 240,0 size 76x30; TextOff 'Text'
      on Release: ActivateScreen("6. DATA E HORA", 0)

screen "1. INÍCIO" 320x240, template "MOURA"
   on GenerateScreen: SetTag("Número da Tela", 1)
   TextField "Text field_7" at 146,38 size 80x15; Text 'STEELBELT'
   TextField "Text field_2" at 144,61 size 85x13; Text 'EM OPERAÇÃO'
   Circle "Circle_2" at 237,60 size 14x14
      Appearance <- "Status_Empastadeira.Em operação"
   TextField "Text field_3" at 144,84 size 85x13; Text 'EMERGÊNCIA'
   Circle "Circle_3" at 237,83 size 14x14
      Appearance <- "Status_Empastadeira.Emergência Ativa"
   TextField "Text field_4" at 144,107 size 85x13; Text 'MANUAL'
   Circle "Circle_4" at 237,106 size 14x14
      Appearance <- "Status_Empastadeira.Manual"
   TextField "Text field_5" at 144,130 size 85x13; Text 'AUTOMÁTICO'
   Circle "Circle_5" at 237,129 size 14x14
      Appearance <- "Status_Empastadeira.Automatico"
   TextField "Text field_6" at 144,153 size 85x13; Text 'COMUNICAÇÃO'
   Circle "Circle_6" at 237,152 size 14x14
      Appearance <- "DB_Controle_Perda Comunicação"
   TextField "Text field_9" at 16,60 size 83x13; Text 'EM OPERAÇÃO'
   Circle "Circle_7" at 108,60 size 14x14
      Appearance <- "Status_Diverger.Em operação"
   TextField "Text field_10" at 16,83 size 83x13; Text 'EMERGÊNCIA'
   Circle "Circle_8" at 108,83 size 14x14
      Appearance <- "Status_Diverger.Emergência Ativa"
   TextField "Text field_11" at 16,106 size 83x13; Text 'MANUAL'
   Circle "Circle_9" at 108,106 size 14x14
      Appearance <- "Status_Diverger.Manual"
   TextField "Text field_12" at 16,130 size 83x13; Text 'AUTOMÁTICO'
   Circle "Circle_10" at 108,129 size 14x14
      Appearance <- "Status_Diverger.Automatico"
   TextField "Text field_1" at 16,153 size 83x13; Text 'FALHA INV 01'
   Circle "Circle_11" at 108,152 size 14x14
      Appearance <- "Status_Diverger.Falha Inv 01"
   TextField "Text field_8" at 16,176 size 83x13; Text 'FALHA INV 02'
   Circle "Circle_1" at 108,175 size 14x14
      Appearance <- "Status_Diverger.Falha Inv 02"
   TextField "Text field_14" at 18,38 size 80x15; Text 'DIVIDER'
   IOField "Velocidade da Linha" at 218,182 size 95x22; FormatPattern 99.9; Unit  m/min
      ProcessValue <- "Status_Velocidade SteelBelt"
   TextField "Txt_VelocidadeLinha" at 146,181 size 69x24; Text 'VELOCIDADE DA LINHA:'
   Button "Botão_Reset" at 271,36 size 38x38; TextOff 'Text'; PictureOff "Reset"
      on Press: SetBit("DB_Controle_Reset Falha")
      on Release: ResetBit("DB_Controle_Reset Falha")
   TextField "Txt_Reset" at 273,71 size 35x15; Text 'Reset'
   Group "DIVIDER" at 8,38 size 122x160
   Group "STEELBELT" at 136,38 size 125x136
   Button "Botão_Ajustes" at 271,88 size 38x38; TextOff 'Text'; PictureOff "Ajustes"
      on Release: ActivateScreen("2. MENU", 0)
   TextField "Txt_Ajustes" at 274,123 size 33x15; Text 'Menu'
   IOField "I/O field_1" at 269,140 size 42x23; FormatPattern 9.999
      ProcessValue <- "Status_Fator %"
   TextField "Txt_Ajustes_1" at 266,161 size 48x15; Text 'Menu / Fator %'

screen "3. VELOCIDADES" 320x240, template "MOURA"
   on GenerateScreen: SetTag("Número da Tela", 3)
   on ClearScreen: ResetBit("Pop-up SPAN"); ResetBit("Pop-up ZERO")
   Softkey "Softkey_F6" at 266,202 size 53x38
      on KeyDown: function_ee5b8808("Popup_SPAN")
      on KeyUp: function_f101fd67("Popup_SPAN")
   Softkey "Softkey_F4" at 160,202 size 53x38
      on KeyDown: function_ee5b8808("Popup_ZERO")
      on KeyUp: function_f101fd67("Popup_ZERO")
   Button "Home" at 148,213 size 25x25; TextOff 'Text'; PictureOff "Início"
      on Release: ActivateScreen("1. INÍCIO", 0)
   Button "Previus" at 3,213 size 25x25; TextOff 'Text'; PictureOff "Left_Arrow_3"
      on Release: function_efd93a16()
   TextField "Barra_InversoresFrequência" at 10,34 size 300x25; Text 'INVERSORES DE FREQUÊNCIA'
   TextField "Barra_DividerDancerSensor" at 10,132 size 300x25; Text 'DIVIDER DANCER SENSOR'
   TextField "Txt_Esteira01" at 10,107 size 75x25; Text 'ESTEIRA 01'
   IOField "Valor_Esteira01" at 85,107 size 75x25; Authorization "User administration"; FormatPattern 99.9; Unit  m/min
      ProcessValue <- "Esteira 01_Speed"
   TextField "Txt_Esteira02" at 160,107 size 75x25; Text 'ESTEIRA 02'
   IOField "Valor_Esteira02" at 235,107 size 75x25; Authorization "User administration"; FormatPattern 99.9; Unit  m/min
      ProcessValue <- "Esteira 02_Speed"
   TextField "Txt_AlturaMalha" at 10,157 size 300x25; Text 'ALTURA DA MALHA SP='
   IOField "Valor_AlturaMalha" at 235,157 size 75x25; Authorization "User administration"; FormatPattern 999.9; Unit  mm
      ProcessValue <- "Sensor_Escalonado"
   TextField "Txt_SteelBelt" at 10,59 size 225x25; Text 'STEELBELT (VELOCIDADE MESTRE)'
   IOField "Valor_SteelBelt" at 235,59 size 75x25; Authorization "User administration"; FormatPattern 99.9; Unit  m/min
      ProcessValue <- "Status_Velocidade SteelBelt"
   TextField " Txt_CalibraçãoSensor" at 10,181 size 300x25; Text 'CALIBRAÇÃO DO SENSOR'
   Button "Popup_SPAN" at 260,181 size 50x25; TextOff 'SPAN'; HelpText 'SPAN = POSICIONE O SENSOR 80MM DO PISO.'
      on Release: SetBit("Pop-up SPAN"); ResetBit("Pop-up ZERO")
   Button "Popup_ZERO" at 161,181 size 50x25; TextOff 'ZERO'; HelpText 'ZERO = POSICIONE O LASER DO SENSOR NO PISO (0MM).'
      on Release: SetBit("Pop-up ZERO"); ResetBit("Pop-up SPAN")
   Button "Botão_SETPOINT" at 210,181 size 50x25; TextOff 'SP'; Authorization "User administration"
      on Release: ResetBit("KEY_MARK")
      on Press: SetBit("KEY_MARK")
   IOField "TempoMáximo_1" at 160,158 size 75x23; Authorization "User administration"; FormatPattern 999.9; Unit  mm
      ProcessValue <- "Check_mark"
   TextField "Txt_Divider" at 10,83 size 225x25; Text 'DIVIDER'
   IOField "Valor_Divider" at 235,83 size 75x25; Authorization "User administration"; FormatPattern 99.9; Unit  m/min
      ProcessValue <- "Divider Speed"
   Softkey "Softkey_F5" at 0,0 size 0x0
      on KeyDown: function_ee5b8808("Botão_SETPOINT")
      on KeyUp: function_f101fd67("Botão_SETPOINT")
   Rectangle "Fundo_SPAN" at 42,63 size 235x120
      Visibility <- "Pop-up SPAN"
   TextField "Barra_SPAN" at 42,63 size 235x25; Text 'CALIBRAR SPAN'
      Visibility <- "Pop-up SPAN"
   Button "Botão_Fechar_SPAN" at 252,63 size 25x25; TextOff 'X'
      Visibility <- "Pop-up SPAN"
      on Release: ResetBit("Pop-up SPAN")
   TextField "Txt_SPAN" at 50,95 size 201x30; Text 'POSICIONE O LASER DO SENSOR A 80MM DO PISO.'
      Visibility <- "Pop-up SPAN"
   TextField "Txt_ValorAnal_SPAN" at 181,126 size 82x13; Text 'Valor analógico:'
      Visibility <- "Pop-up SPAN"
   Button "Botão_SPAN" at 53,145 size 90x25; HelpText 'SPAN = POSICIONE O SENSOR 80MM DO PISO.'; TextOff 'SPAN'; Authorization "User administration"
      on Release: ResetBit("KEY_SPAN")
      on Press: SetBit("KEY_SPAN")
      Visibility <- "Pop-up SPAN"
   IOField "Valor_SPAN" at 177,145 size 90x25; Authorization "User administration"; FormatPattern 99999
      ProcessValue <- "Divider Dancer.X1"
      Visibility <- "Pop-up SPAN"
   Group "Grupo_SPAN" at 42,63 size 235x120
   Rectangle "Fundo_ZERO" at 42,63 size 235x120
      Visibility <- "Pop-up ZERO"
   TextField "Barra_ZERO" at 42,63 size 235x25; Text 'CALIBRAR ZERO'
      Visibility <- "Pop-up ZERO"
   Button "Botão_Fechar_ZERO" at 252,63 size 25x25; TextOff 'X'
      Visibility <- "Pop-up ZERO"
      on Release: ResetBit("Pop-up ZERO")
   TextField "Txt_ZERO" at 50,95 size 201x30; Text 'POSICIONE O LASER DO SENSOR NO PISO (0MM).'
      Visibility <- "Pop-up ZERO"
   TextField "Txt_ValorAnal_ZERO" at 181,126 size 82x13; Text 'Valor analógico:'
      Visibility <- "Pop-up ZERO"
   Button "Botão_ZERO" at 53,145 size 90x25; HelpText 'SPAN = POSICIONE O SENSOR 80MM DO PISO.'; TextOff 'ZERO'; Authorization "User administration"
      Visibility <- "Pop-up ZERO"
      on Release: ResetBit("KEY_ZERO")
      on Press: SetBit("KEY_ZERO")
   IOField "Valor_ZERO" at 177,145 size 90x25; Authorization "User administration"; FormatPattern 99999
      Visibility <- "Pop-up ZERO"
      ProcessValue <- "Divider Dancer.X0"
   Group "Grupo_ZERO" at 42,63 size 235x120

screen "2. MENU" 320x240, template "MOURA"
   on GenerateScreen: SetTag("Número da Tela", 2)
   Softkey "Softkey_F5" at 213,202 size 53x38
      on KeyUp: function_f101fd67("Painel de Controle")
      on KeyDown: function_ee5b8808("Painel de Controle")
   Softkey "Softkey_F4" at 160,202 size 53x38
      on KeyUp: function_f101fd67("Ajutar Data/Hora")
      on KeyDown: function_ee5b8808("Ajutar Data/Hora")
   Button "Tempos" at 76,40 size 170x25; TextOff 'VELOCIDADES (F1)'
      on Release: ActivateScreen("3. VELOCIDADES", 0)
   Button "Home" at 148,213 size 25x25; TextOff 'Text'; PictureOff "Início"
      on Release: ActivateScreen("1. INÍCIO", 0)
   Button "Entradas Digitais" at 76,73 size 170x25; TextOff 'ENTRADAS DIGITAIS (F2)'
      on Release: ActivateScreen("4. ENTRADAS", 0)
   Button "Saídas Digitais" at 76,107 size 170x25; TextOff 'SAÍDAS DIGITAIS (F3)'
      on Release: ActivateScreen("5. SAÍDAS", 0)
   Button "Painel de Controle" at 76,175 size 170x25; TextOff 'PAINEL DE CONTROLE (F5)'; Authorization "User administration"
      on Release: StopRuntime(0)
   Button "Ajutar Data/Hora" at 76,141 size 170x25; TextOff 'AJUSTAR DATA/HORA (F4)'
      on Release: ActivateScreen("6. DATA E HORA", 0)
   Button "Botão_Logon" at 265,40 size 38x38; TextOff 'Text'; PictureOff "LOGON"
      on Release: function_a2a04561()
   Button "Botão_Logoff" at 265,81 size 38x38; TextOff 'Text'; PictureOff "LOGOFF"
      on Release: function_f23ef4c9()
   Softkey "Softkey_F1" at 0,0 size 0x0
      on KeyDown: function_ee5b8808("Tempos")
      on KeyUp: function_f101fd67("Tempos")
   Softkey "Softkey_F2" at 0,0 size 0x0
      on KeyDown: function_ee5b8808("Entradas Digitais")
      on KeyUp: function_f101fd67("Entradas Digitais")
   Softkey "Softkey_F3" at 0,0 size 0x0
      on KeyDown: function_ee5b8808("Saídas Digitais")
      on KeyUp: function_f101fd67("Saídas Digitais")

screen "4. ENTRADAS" 320x240, template "MOURA"
   on GenerateScreen: SetTag("Número da Tela", 4)
   Button "Home" at 148,213 size 25x25; TextOff 'Text'; PictureOff "Início"
      on Release: ActivateScreen("1. INÍCIO", 0)
   TextField "Emergência" at 1,34 size 160x20; Text 'I0.0 - MAN / AUTO'
   Circle "Emergência Circle" at 145,38 size 12x12
      Appearance <- "I0.0 - MAN / AUTO"
   TextField "Reset" at 1,53 size 160x20; Text 'I0.1 - VFD 01 MANUAL'
   TextField "Manual" at 1,72 size 160x20; Text 'I0.2 - VFD 02 MANUAL'
   TextField "Automático" at 1,91 size 160x20; Text 'I0.3 - EMERGÊNCIA'
   TextField "Ciclo Automático" at 1,110 size 160x20; Text 'I0.4 - LIGA / DESLIGA'
   TextField "Oxigênio" at 1,129 size 160x20; Text 'I0.5 - FALHA VFD 01'
   TextField "Sensor Entrada" at 1,148 size 160x20; Text 'I0.6 - FALHA VFD 02'
   TextField "Sensor Workstation" at 1,167 size 160x20; Text 'I0.7 - BOTÃO JOG'
   TextField "Cabeçote Avançado" at 1,186 size 160x20; Text 'I1.0 - RESERVA'
   TextField "Cabeçote Recuado" at 160,34 size 160x20; Text 'I1.1 - RESERVA'
   Circle "Reset Circle" at 145,57 size 12x12
      Appearance <- "I0.1 - VFD 01 MANUAL"
   Circle "Manual Circle" at 145,76 size 12x12
      Appearance <- "I0.2 - VFD 02 MANUAL"
   Circle "Automático Circle" at 145,95 size 12x12
      Appearance <- "I0.3 - EMERGÊNCIA"
   Circle "Ciclo Automático Circle" at 145,114 size 12x12
      Appearance <- "I0.4 - LIGA / DESLIGA"
   Circle "Oxigênio Circle" at 145,133 size 12x12
      Appearance <- "I0.5 - FALHA VFD 01"
   Circle "Sensor Entrada Circle" at 145,152 size 12x12
      Appearance <- "I0.6 - FALHA VFD 02"
   Circle "Sensor Workstation Circle" at 145,171 size 12x12
      Appearance <- "I0.7 - BOTÃO JOG"
   Circle "Cabeçote Avançado Circle" at 145,190 size 12x12
      Appearance <- "Sempre_0"
   TextField "Esteira_10" at 160,53 size 160x20; Text 'I1.2 - RESERVA'
   TextField "Eletrodo Recuado" at 160,72 size 160x20; Text 'I1.3 - RESERVA'
   TextField "Fluxostato Direito" at 160,91 size 160x20; Text 'I1.4 - RESERVA'
   TextField "Fluxostato Esquerdo" at 160,110 size 160x20; Text 'I1.5 - RESERVA'
   TextField "Baixa Temp. Direita" at 160,129 size 160x20; Text '- - - - -'
   TextField "Baixa Temp. Esquerda" at 160,148 size 160x20; Text '- - - - -'
   TextField "Alta Temp. Direita" at 160,167 size 160x20; Text '- - - - -'
   TextField "Alta Temp. Esquerda" at 160,186 size 160x20; Text '- - - - -'
   Circle "Cabeçote Recuado Circle" at 304,38 size 12x12
      Appearance <- "Sempre_0"
   Circle "Circle_11" at 304,57 size 12x12
      Appearance <- "Sempre_0"
   Circle "Eletrodo Recuado Circle" at 304,76 size 12x12
      Appearance <- "Sempre_0"
   Circle "Fluxostato Direito Circle" at 304,95 size 12x12
      Appearance <- "Sempre_0"
   Circle "Fluxostato Esquerdo Circle" at 304,114 size 12x12
      Appearance <- "Sempre_0"
   Button "Previus" at 3,213 size 25x25; TextOff 'Text'; PictureOff "Left_Arrow_1"
      on Release: function_efd93a16()

screen "6. DATA E HORA" 320x240, template "MOURA"
   on GenerateScreen: SetTag("Número da Tela", 6)
   Button "Home" at 148,213 size 25x25; TextOff 'Text'; PictureOff "Início"
      on Release: ActivateScreen("1. INÍCIO", 0)
   TextField ""DATA"" at 11,77 size 200x25; Text 'DATA'
   TextField ""HORA"" at 210,77 size 100x25; Text 'HORA'
   IOField "Dia" at 16,107 size 46x18; FormatPattern 99; Unit   de
      ProcessValue <- "Dia"
   IOField "Ano" at 165,107 size 39x18; FormatPattern 9999
      ProcessValue <- "Ano"
   SymbolicIOField "Mês" at 65,106 size 74x20; TextOn '1'; TextOff '0'; TextList "Mês"
      ProcessValue <- "Mês"
   TextField ""de"" at 142,107 size 20x18; Text 'de'
   IOField "Minuto" at 249,107 size 31x18; FormatPattern 99; Unit  :
      ProcessValue <- "Minuto"
   IOField "Hora" at 218,107 size 31x18; FormatPattern 99; Unit  :
      ProcessValue <- "Hora"
   IOField "Segundo" at 280,107 size 23x18; FormatPattern 99
      ProcessValue <- "Segundo"
   Button "Salvar" at 220,136 size 90x25; TextOff 'SALVAR (F6)'
      on Release: ResetBit("Editar_Data_Hora")
      on Press: SetBit("Editar_Data_Hora")
   Button "Previus" at 3,213 size 25x25; TextOff 'Text'; PictureOff "Left_Arrow_2"
      on Release: function_efd93a16()
   Softkey "Softkey_F6" at 266,202 size 53x38
      on KeyUp: function_f101fd67("Salvar")
      on KeyDown: function_ee5b8808("Salvar")

screen "5. SAÍDAS" 320x240, template "MOURA"
   on GenerateScreen: SetTag("Número da Tela", 5)
   Button "Home" at 148,213 size 25x25; TextOff 'Text'; PictureOff "Início"
      on Release: ActivateScreen("1. INÍCIO", 0)
   TextField "Q0.0" at 1,34 size 160x20; Text 'Q0.0 - LIGA VFD 01'
   Circle "Circle Q0.0" at 145,38 size 12x12
      Appearance <- "Q0.0 - LIGA VFD 01"
   TextField "Q0.1" at 1,53 size 160x20; Text 'Q0.1 - LIGA VFD 02'
   TextField "Q0.4" at 1,110 size 160x20; Text 'Q0.4 - LIGA VFD DIVIDER'
   TextField "Q0.5" at 1,129 size 160x20; Text 'Q0.5 - RESERVA'
   TextField "Q0.6" at 1,148 size 160x20; Text 'Q0.6 - RESERVA'
   TextField "Q0.7" at 1,167 size 160x20; Text 'Q0.7 - RESERVA'
   TextField "Q1.0" at 1,186 size 160x20; Text 'Q1.0 - RESERVA'
   TextField "Q1.1" at 160,34 size 160x20; Text 'Q1.1 - RESERVA'
   Circle "Circle Q0.1" at 145,57 size 12x12
      Appearance <- "Q0.1 - LIGA VFD 02"
   Circle "Circle Q0.4" at 145,114 size 12x12
      Appearance <- "Q0.4 - LIGA VFD DIVIDER"
   Circle "Circle Q0.5" at 145,133 size 12x12
      Appearance <- "Sempre_0"
   Circle "Circle Q0.6" at 145,152 size 12x12
      Appearance <- "Sempre_0"
   Circle "Circle Q0.7" at 145,171 size 12x12
      Appearance <- "Sempre_0"
   Circle "Circle Q01.0" at 145,190 size 12x12
      Appearance <- "Sempre_0"
   TextField "Empty1" at 160,53 size 160x20; Text '- - - - -'
   TextField "Empty2" at 160,72 size 160x20; Text '- - - - -'
   TextField "Empty3" at 160,91 size 160x20; Text '- - - - -'
   TextField "Empty4" at 160,110 size 160x20; Text '- - - - -'
   TextField "Empty5" at 160,129 size 160x20; Text '- - - - -'
   TextField "Empty6" at 160,148 size 160x20; Text '- - - - -'
   TextField "Empty7" at 160,167 size 160x20; Text '- - - - -'
   TextField "Empty8" at 160,186 size 160x20; Text '- - - - -'
   Circle "Circle Q1.1" at 304,38 size 12x12
      Appearance <- "Sempre_0"
   Button "Previus" at 3,213 size 25x25; TextOff 'Text'; PictureOff "Left_Arrow_3"
      on Release: function_efd93a16()
   Group "Group" at 0,72 size 161x39
   TextField "Text field_1" at 247,214 size 68x24; Text '* Clique para resetar'
   TextField "Q0.2" at 1,72 size 160x20; Text 'Q0.2 - RESET VFD 01 *'
   Circle "Circle Q0.2" at 145,76 size 12x12
      Appearance <- "Q0.2 - RESET VFD 01"
   TextField "Q0.3" at 1,91 size 160x20; Text 'Q0.3 - RESET VFD 02 *'
   Circle "Circle Q0.3" at 145,95 size 12x12
      Appearance <- "Q0.3 - RESET VFD 02"
   Button "Botão_Reset" at 0,73 size 160x38; TextOff 'Text'

scheduled task "Sempre_0"
   on Action: SetTag("Sempre_0", 0)
*)